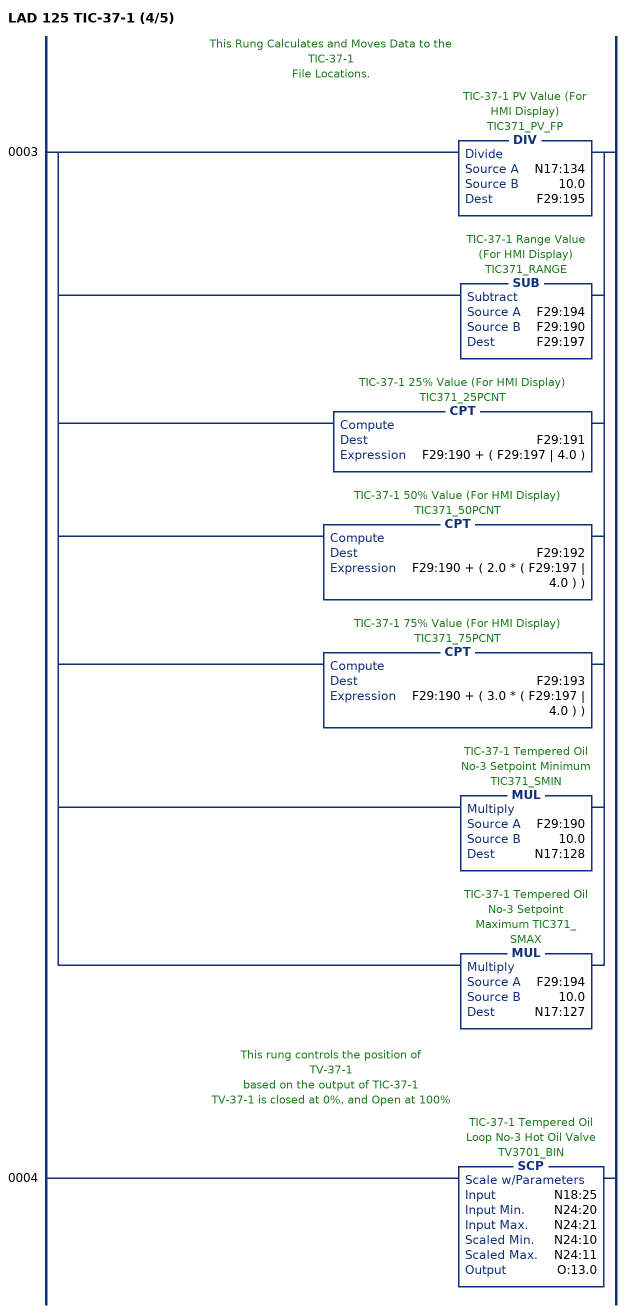
% Rung: 3 %
% This Rung Calculates and Moves Data to the
% TIC-37-1
% File Locations. %
SOR BST DIV N17:134 10.0 F29:195 NXB SUB F29:194 F29:190 F29:197 NXB CPT F29:191 " F29:190 + ( F29:197 | 4.0 ) " NXB CPT F29:192 " F29:190 + ( 2.0 * ( F29:197 | 4.0 ) ) " NXB CPT F29:193 " F29:190 + ( 3.0 * ( F29:197 | 4.0 ) ) " NXB MUL F29:190 10.0 N17:128 NXB MUL F29:194 10.0 N17:127 BND EOR
%   N17:134  TIC371_PV  "TIC-37-1 Tempered Oil No-3 Scaled Process Variable" %
%   F29:195  TIC371_PV_FP  "TIC-37-1 PV Value (For HMI Display)" %
%   F29:194  TIC371_MAX  "TIC-37-1 100% Value (For HMI Display)" %
%   F29:190  TIC371_MIN  "TIC-37-1 0% Value (For HMI Display)" %
%   F29:197  TIC371_RANGE  "TIC-37-1 Range Value (For HMI Display)" %
%   F29:191  TIC371_25PCNT  "TIC-37-1 25% Value (For HMI Display)" %
%   F29:192  TIC371_50PCNT  "TIC-37-1 50% Value (For HMI Display)" %
%   F29:193  TIC371_75PCNT  "TIC-37-1 75% Value (For HMI Display)" %
%   N17:128  TIC371_SMIN  "TIC-37-1 Tempered Oil No-3 Setpoint Minimum" %
%   N17:127  TIC371_SMAX  "TIC-37-1 Tempered Oil No-3 Setpoint Maximum" %
% Rung: 4 %
% This rung controls the position of
% TV-37-1
% based on the output of TIC-37-1
% TV-37-1 is closed at 0%, and Open at 100% %
SOR SCP N18:25 N24:20 N24:21 N24:10 N24:11 O:13.0 EOR
%   N18:25  TIC371_OUT1  "TIC-37-1 Tempered Oil No-3 PID Output Value" %
%   N24:20  PID_MIN  "PID Statement Minimum Value" %
%   N24:21  PID_MAX  "PID Statement Maximum Value" %
%   N24:10  AO_MIN_NO4I  "Analog Output Minimum Value Generates 4 mA DC (To NO4I AO Module)" %
%   N24:11  AO_MAX_NO4I  "Analog Output Maximum Value Generates 20 mA DC (To NO4I AO Module)" %
%   O:13.0  TV3701_BIN  "TIC-37-1 Tempered Oil Loop No-3 Hot Oil Valve" %

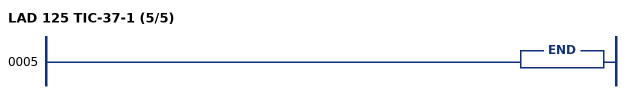
% Rung: 5 %
SOR END EOR

LADDER 126 "TIC-40-1"    % Tempered Oil Loop No-2 Temperature PID Controls %
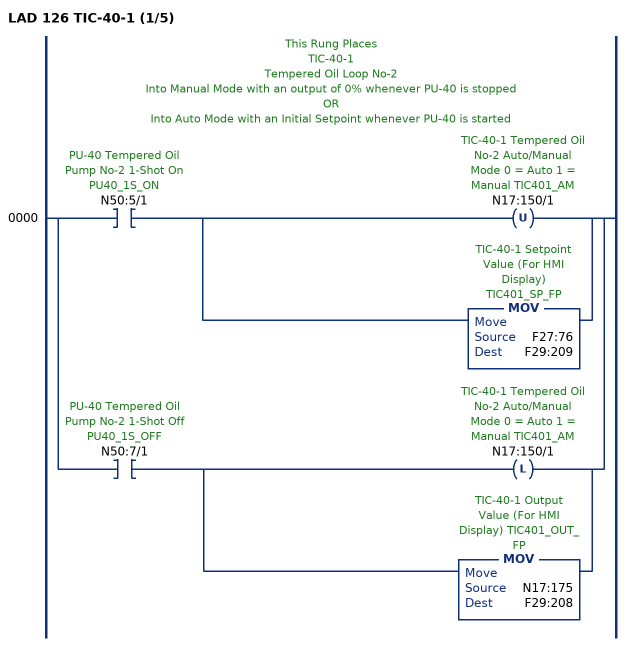
% Rung: 0 %
% This Rung Places
% TIC-40-1
% Tempered Oil Loop No-2
% Into Manual Mode with an output of 0% whenever PU-40 is stopped
% OR
% Into Auto Mode with an Initial Setpoint whenever PU-40 is started %
SOR BST XIC N50:5/1 BST OTU N17:150/1 NXB MOV F27:76 F29:209 BND NXB XIC N50:7/1 BST OTL N17:150/1 NXB MOV N17:175 F29:208 BND BND EOR
%   N50:5/1  PU40_1S_ON  "PU-40 Tempered Oil Pump No-2 1-Shot On" %
%   N17:150/1  TIC401_AM  "TIC-40-1 Tempered Oil No-2 Auto/Manual Mode 0 = Auto 1 = Manual" %
%   F27:76  TIC401_INIT_SP  "TIC-40-1 Initial Temperature Setpoint" %
%   F29:209  TIC401_SP_FP  "TIC-40-1 Setpoint Value (For HMI Display)" %
%   N50:7/1  PU40_1S_OFF  "PU-40 Tempered Oil Pump No-2 1-Shot Off" %
%   N17:175  TIC401_OFF_OUTPUT  "TIC-40-1 Output When PU-13 Is Off" %
%   F29:208  TIC401_OUT_FP  "TIC-40-1 Output Value (For HMI Display)" %

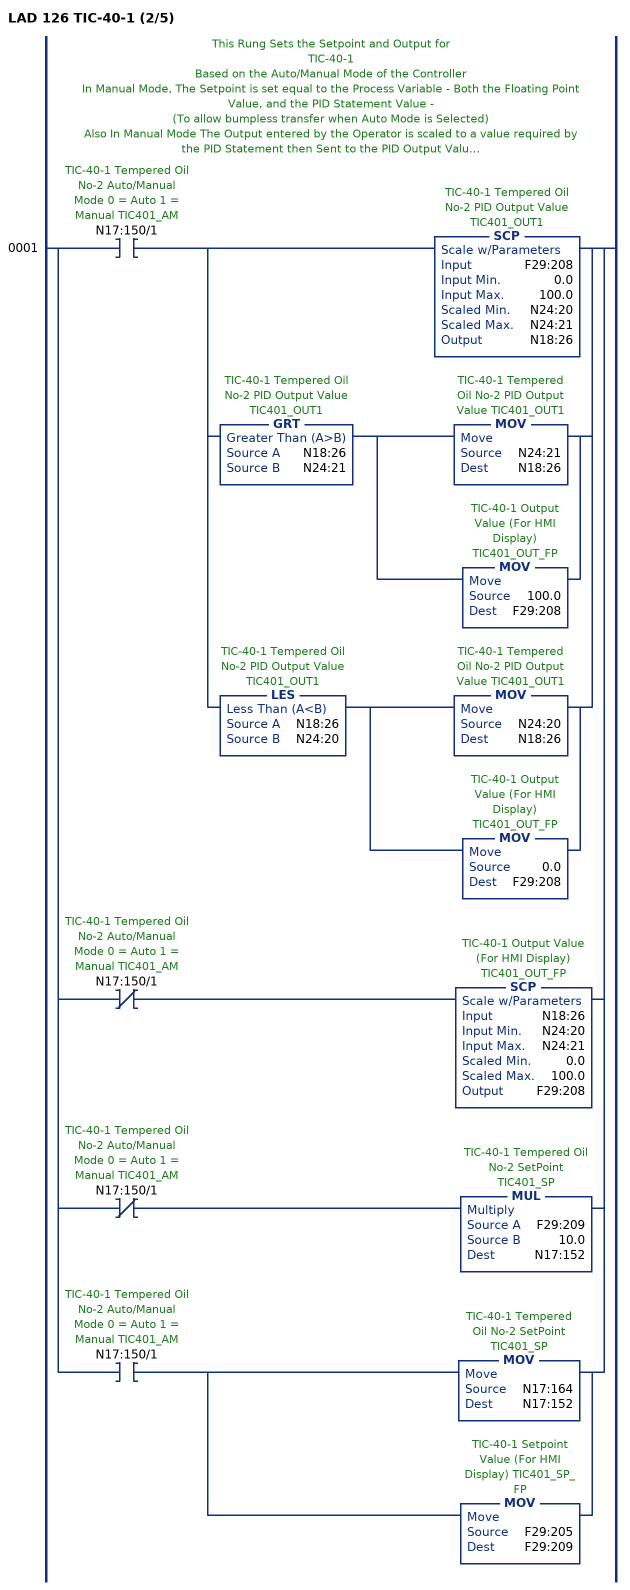
% Rung: 1 %
% This Rung Sets the Setpoint and Output for
% TIC-40-1
% Based on the Auto/Manual Mode of the Controller
% In Manual Mode, The Setpoint is set equal to the Process Variable - Both the Floating Point Value, and the PID Statement Value -
% (To allow bumpless transfer when Auto Mode is Selected)
% Also In Manual Mode The Output entered by the Operator is scaled to a value required by the PID Statement then Sent to the PID Output Value
% 
% In Auto Mode, The Setpoint is Entered by the Operator from Any HMI terminal, Multiplied by 10, and placed in the PID Statement's Setpoint Location
% Also In Auto Mode, the Output (used by the Operator) is set equal to the actual value of the pID statement
% (To allow bumpless transfer when Manual Mode is Selected) %
SOR BST XIC N17:150/1 BST SCP F29:208 0.0 100.0 N24:20 N24:21 N18:26 NXB GRT N18:26 N24:21 BST MOV N24:21 N18:26 NXB MOV 100.0 F29:208 BND NXB LES N18:26 N24:20 BST MOV N24:20 N18:26 NXB MOV 0.0 F29:208 BND BND NXB XIO N17:150/1 SCP N18:26 N24:20 N24:21 0.0 100.0 F29:208 NXB XIO N17:150/1 MUL F29:209 10.0 N17:152 NXB XIC N17:150/1 BST MOV N17:164 N17:152 NXB MOV F29:205 F29:209 BND BND EOR
%   N17:150/1  TIC401_AM  "TIC-40-1 Tempered Oil No-2 Auto/Manual Mode 0 = Auto 1 = Manual" %
%   F29:208  TIC401_OUT_FP  "TIC-40-1 Output Value (For HMI Display)" %
%   N24:20  PID_MIN  "PID Statement Minimum Value" %
%   N24:21  PID_MAX  "PID Statement Maximum Value" %
%   N18:26  TIC401_OUT1  "TIC-40-1 Tempered Oil No-2 PID Output Value" %
%   F29:209  TIC401_SP_FP  "TIC-40-1 Setpoint Value (For HMI Display)" %
%   N17:152  TIC401_SP  "TIC-40-1 Tempered Oil No-2 SetPoint" %
%   N17:164  TIC401_PV  "TIC-40-1 Tempered Oil No-2 Scaled Process Variable" %
%   F29:205  TIC401_PV_FP  "TIC-40-1 PV Value (For HMI Display)" %

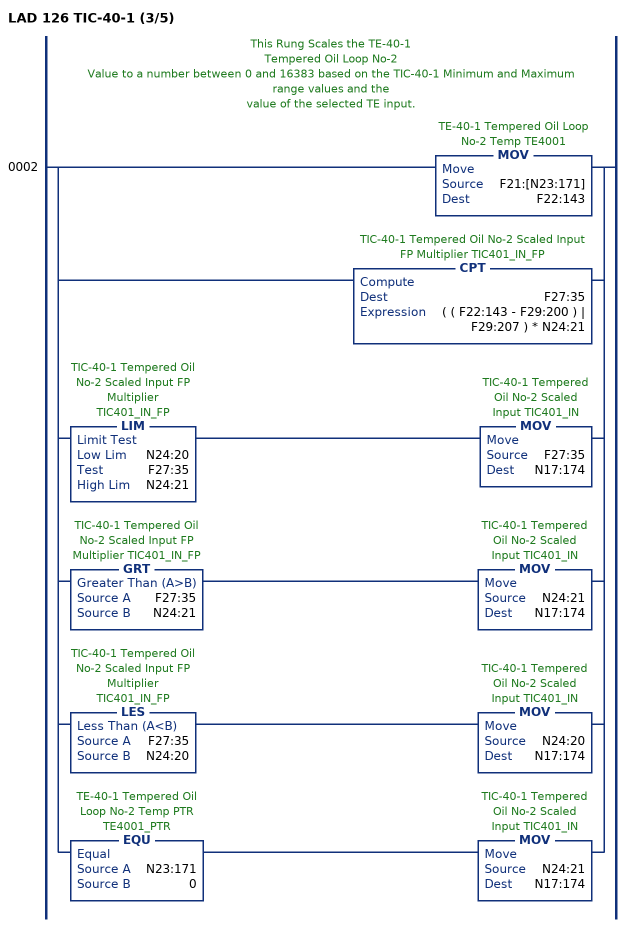
% Rung: 2 %
% This Rung Scales the TE-40-1
% Tempered Oil Loop No-2
% Value to a number between 0 and 16383 based on the TIC-40-1 Minimum and Maximum range values and the
% value of the selected TE input. %
SOR BST MOV F21:[N23:171] F22:143 NXB CPT F27:35 " ( ( F22:143 - F29:200 ) | F29:207 ) * N24:21 " NXB LIM N24:20 F27:35 N24:21 MOV F27:35 N17:174 NXB GRT F27:35 N24:21 MOV N24:21 N17:174 NXB LES F27:35 N24:20 MOV N24:20 N17:174 NXB EQU N23:171 0 MOV N24:21 N17:174 BND EOR
%   N23:171  TE4001_PTR  "TE-40-1 Tempered Oil Loop No-2 Temp PTR" %
%   F22:143  TE4001  "TE-40-1 Tempered Oil Loop No-2 Temp" %
%   F27:35  TIC401_IN_FP  "TIC-40-1 Tempered Oil No-2 Scaled Input FP Multiplier" %
%   F29:200  TIC401_MIN  "TIC-40-1 0% Value (For HMI Display)" %
%   F29:207  TIC401_RANGE  "TIC-40-1 Range Value (For HMI Display)" %
%   N24:21  PID_MAX  "PID Statement Maximum Value" %
%   N24:20  PID_MIN  "PID Statement Minimum Value" %
%   N17:174  TIC401_IN  "TIC-40-1 Tempered Oil No-2 Scaled Input" %

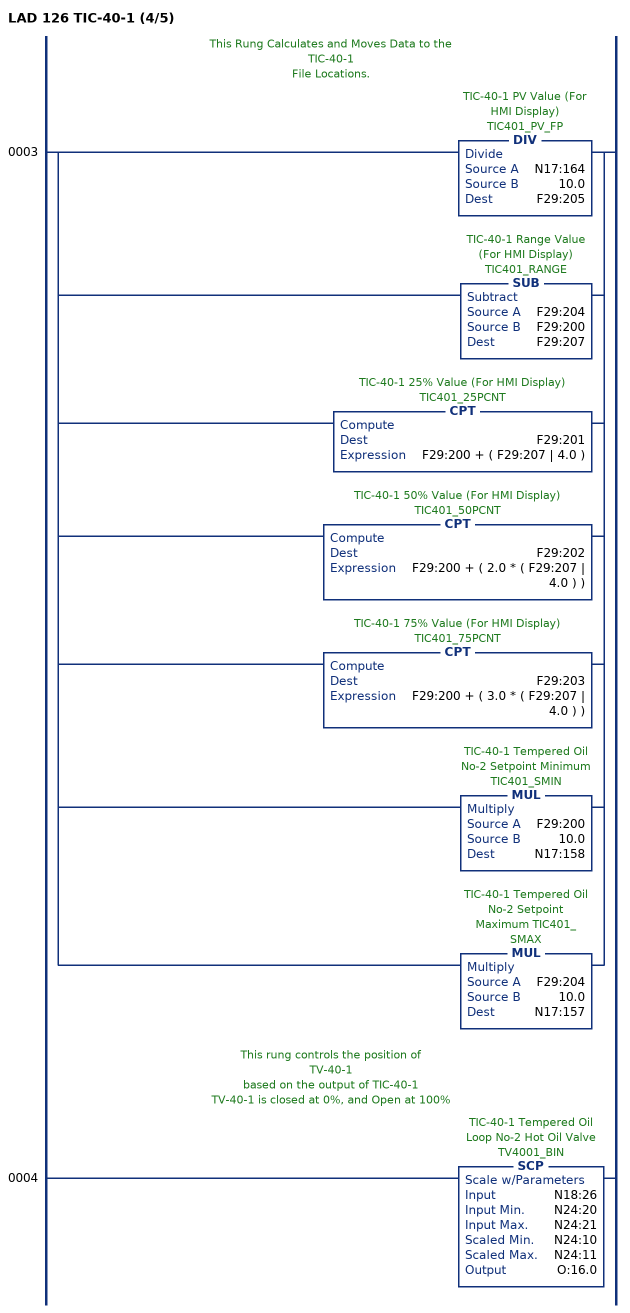
% Rung: 3 %
% This Rung Calculates and Moves Data to the
% TIC-40-1
% File Locations. %
SOR BST DIV N17:164 10.0 F29:205 NXB SUB F29:204 F29:200 F29:207 NXB CPT F29:201 " F29:200 + ( F29:207 | 4.0 ) " NXB CPT F29:202 " F29:200 + ( 2.0 * ( F29:207 | 4.0 ) ) " NXB CPT F29:203 " F29:200 + ( 3.0 * ( F29:207 | 4.0 ) ) " NXB MUL F29:200 10.0 N17:158 NXB MUL F29:204 10.0 N17:157 BND EOR
%   N17:164  TIC401_PV  "TIC-40-1 Tempered Oil No-2 Scaled Process Variable" %
%   F29:205  TIC401_PV_FP  "TIC-40-1 PV Value (For HMI Display)" %
%   F29:204  TIC401_MAX  "TIC-40-1 100% Value (For HMI Display)" %
%   F29:200  TIC401_MIN  "TIC-40-1 0% Value (For HMI Display)" %
%   F29:207  TIC401_RANGE  "TIC-40-1 Range Value (For HMI Display)" %
%   F29:201  TIC401_25PCNT  "TIC-40-1 25% Value (For HMI Display)" %
%   F29:202  TIC401_50PCNT  "TIC-40-1 50% Value (For HMI Display)" %
%   F29:203  TIC401_75PCNT  "TIC-40-1 75% Value (For HMI Display)" %
%   N17:158  TIC401_SMIN  "TIC-40-1 Tempered Oil No-2 Setpoint Minimum" %
%   N17:157  TIC401_SMAX  "TIC-40-1 Tempered Oil No-2 Setpoint Maximum" %
% Rung: 4 %
% This rung controls the position of
% TV-40-1
% based on the output of TIC-40-1
% TV-40-1 is closed at 0%, and Open at 100% %
SOR SCP N18:26 N24:20 N24:21 N24:10 N24:11 O:16.0 EOR
%   N18:26  TIC401_OUT1  "TIC-40-1 Tempered Oil No-2 PID Output Value" %
%   N24:20  PID_MIN  "PID Statement Minimum Value" %
%   N24:21  PID_MAX  "PID Statement Maximum Value" %
%   N24:10  AO_MIN_NO4I  "Analog Output Minimum Value Generates 4 mA DC (To NO4I AO Module)" %
%   N24:11  AO_MAX_NO4I  "Analog Output Maximum Value Generates 20 mA DC (To NO4I AO Module)" %
%   O:16.0  TV4001_BIN  "TIC-40-1 Tempered Oil Loop No-2 Hot Oil Valve" %

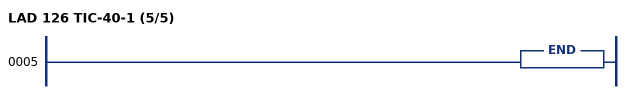
% Rung: 5 %
SOR END EOR

LADDER 131 "LIC-22-1"    % Level Control No-1 PID Controls %
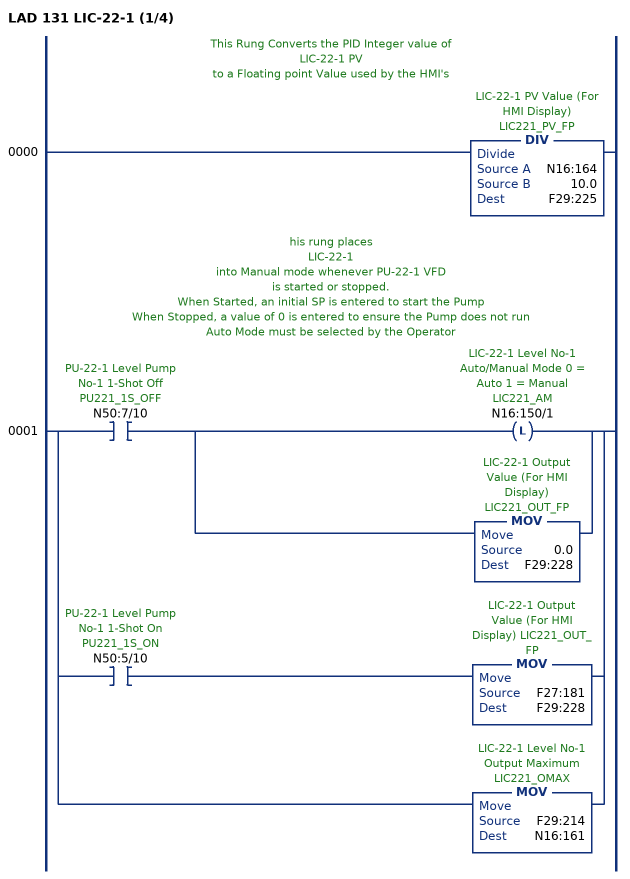
% Rung: 0 %
% This Rung Converts the PID Integer value of
% LIC-22-1 PV
% to a Floating point Value used by the HMI's %
SOR DIV N16:164 10.0 F29:225 EOR
%   N16:164  LIC221_PV  "LIC-22-1 Level No-1 Scaled Process Variable" %
%   F29:225  LIC221_PV_FP  "LIC-22-1 PV Value (For HMI Display)" %
% Rung: 1 %
% his rung places
% LIC-22-1
% into Manual mode whenever PU-22-1 VFD
% is started or stopped.
% When Started, an initial SP is entered to start the Pump
% When Stopped, a value of 0 is entered to ensure the Pump does not run
% Auto Mode must be selected by the Operator %
SOR BST XIC N50:7/10 BST OTL N16:150/1 NXB MOV 0.0 F29:228 BND NXB XIC N50:5/10 MOV F27:181 F29:228 NXB MOV F29:214 N16:161 BND EOR
%   N50:7/10  PU221_1S_OFF  "PU-22-1 Level Pump No-1 1-Shot Off" %
%   N16:150/1  LIC221_AM  "LIC-22-1 Level No-1 Auto/Manual Mode 0 = Auto 1 = Manual" %
%   F29:228  LIC221_OUT_FP  "LIC-22-1 Output Value (For HMI Display)" %
%   N50:5/10  PU221_1S_ON  "PU-22-1 Level Pump No-1 1-Shot On" %
%   F27:181  SIC221_INIT_SP  "SIC-22-1 Initial Speed Setpoint (Hz)" %
%   F29:214  SIC221_MAX  "SIC-22-1 PU-22-1 Level Pump No-1 Freq at 100% Value (For HMI Display)" %
%   N16:161  LIC221_OMAX  "LIC-22-1 Level No-1 Output Maximum" %

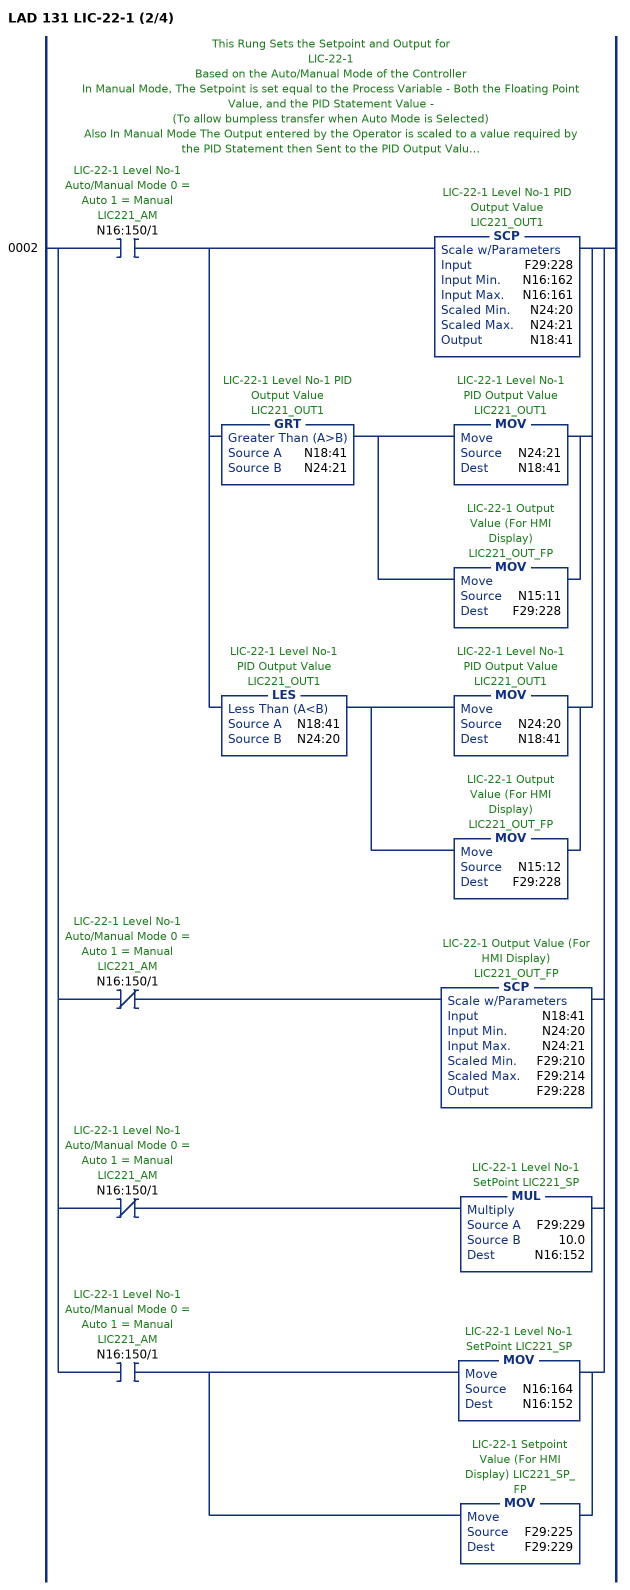
% Rung: 2 %
% This Rung Sets the Setpoint and Output for
% LIC-22-1
% Based on the Auto/Manual Mode of the Controller
% In Manual Mode, The Setpoint is set equal to the Process Variable - Both the Floating Point Value, and the PID Statement Value -
% (To allow bumpless transfer when Auto Mode is Selected)
% Also In Manual Mode The Output entered by the Operator is scaled to a value required by the PID Statement then Sent to the PID Output Value
% 
% In Auto Mode, The Setpoint is Entered by the Operator from Any HMI terminal, Multiplied by 10, and placed in the PID Statement's Setpoint Location
% Also In Auto Mode, the Output (used by the Operator) is set equal to the actual value of the pID statement
% (To allow bumpless transfer when Manual Mode is Selected) %
SOR BST XIC N16:150/1 BST SCP F29:228 N16:162 N16:161 N24:20 N24:21 N18:41 NXB GRT N18:41 N24:21 BST MOV N24:21 N18:41 NXB MOV N15:11 F29:228 BND NXB LES N18:41 N24:20 BST MOV N24:20 N18:41 NXB MOV N15:12 F29:228 BND BND NXB XIO N16:150/1 SCP N18:41 N24:20 N24:21 F29:210 F29:214 F29:228 NXB XIO N16:150/1 MUL F29:229 10.0 N16:152 NXB XIC N16:150/1 BST MOV N16:164 N16:152 NXB MOV F29:225 F29:229 BND BND EOR
%   N16:150/1  LIC221_AM  "LIC-22-1 Level No-1 Auto/Manual Mode 0 = Auto 1 = Manual" %
%   F29:228  LIC221_OUT_FP  "LIC-22-1 Output Value (For HMI Display)" %
%   N16:162  LIC221_OMIN  "LIC-22-1 Level No-1 Output Minimum" %
%   N16:161  LIC221_OMAX  "LIC-22-1 Level No-1 Output Maximum" %
%   N24:20  PID_MIN  "PID Statement Minimum Value" %
%   N24:21  PID_MAX  "PID Statement Maximum Value" %
%   N18:41  LIC221_OUT1  "LIC-22-1 Level No-1 PID Output Value" %
%   N15:11  FIC211_OMAX  "FIC-21-1 Feed Flow No-1 Output Maximum" %
%   N15:12  FIC211_OMIN  "FIC-21-1 Feed Flow No-1 Output Minimum" %
%   F29:210  SIC221_MIN  "SIC-22-1 PU-22-1 Level Pump No-1 Speed 0% Value (For HMI Display)" %
%   F29:214  SIC221_MAX  "SIC-22-1 PU-22-1 Level Pump No-1 Freq at 100% Value (For HMI Display)" %
%   F29:229  LIC221_SP_FP  "LIC-22-1 Setpoint Value (For HMI Display)" %
%   N16:152  LIC221_SP  "LIC-22-1 Level No-1 SetPoint" %
%   N16:164  LIC221_PV  "LIC-22-1 Level No-1 Scaled Process Variable" %
%   F29:225  LIC221_PV_FP  "LIC-22-1 PV Value (For HMI Display)" %

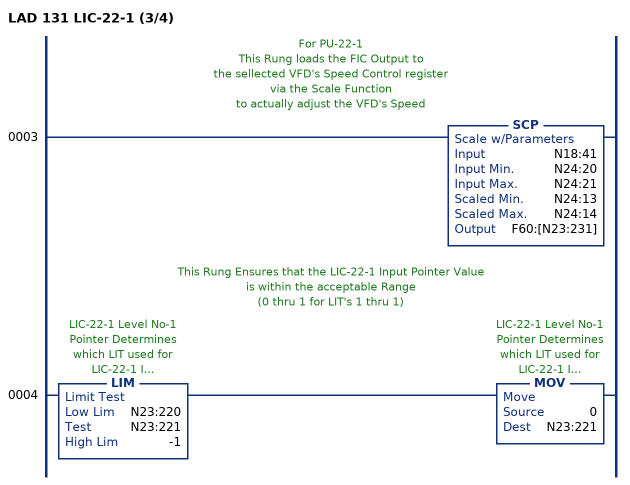
% Rung: 3 %
% For PU-22-1
% This Rung loads the FIC Output to
% the sellected VFD's Speed Control register
% via the Scale Function
% to actually adjust the VFD's Speed %
SOR SCP N18:41 N24:20 N24:21 N24:13 N24:14 F60:[N23:231] EOR
%   N18:41  LIC221_OUT1  "LIC-22-1 Level No-1 PID Output Value" %
%   N24:20  PID_MIN  "PID Statement Minimum Value" %
%   N24:21  PID_MAX  "PID Statement Maximum Value" %
%   N24:13  AO_MIN_OE4  "Analog Output Minimum Value Generates 4 mA DC (To OE4 AO Module)" %
%   N24:14  AO_MAX_OE4  "Analog Output Maximum Value Generates 20 mA DC (To OE4 AO Module)" %
%   N23:231  LIC221_OUT_PTR  "LIC-22-1 Level No-1 Output Pointer Determines which VFD is controled by LIC" %
% Rung: 4 %
% This Rung Ensures that the LIC-22-1 Input Pointer Value
% is within the acceptable Range
% (0 thru 1 for LIT's 1 thru 1) %
SOR LIM N23:220 N23:221 -1 MOV 0 N23:221 EOR
%   N23:220  MAX_LIT_ALLOWED_1  "Maximum Number of LITs Available Plus 1" %
%   N23:221  LIC221_IN_PTR  "LIC-22-1 Level No-1 Pointer Determines which LIT used for LIC-22-1 In" %

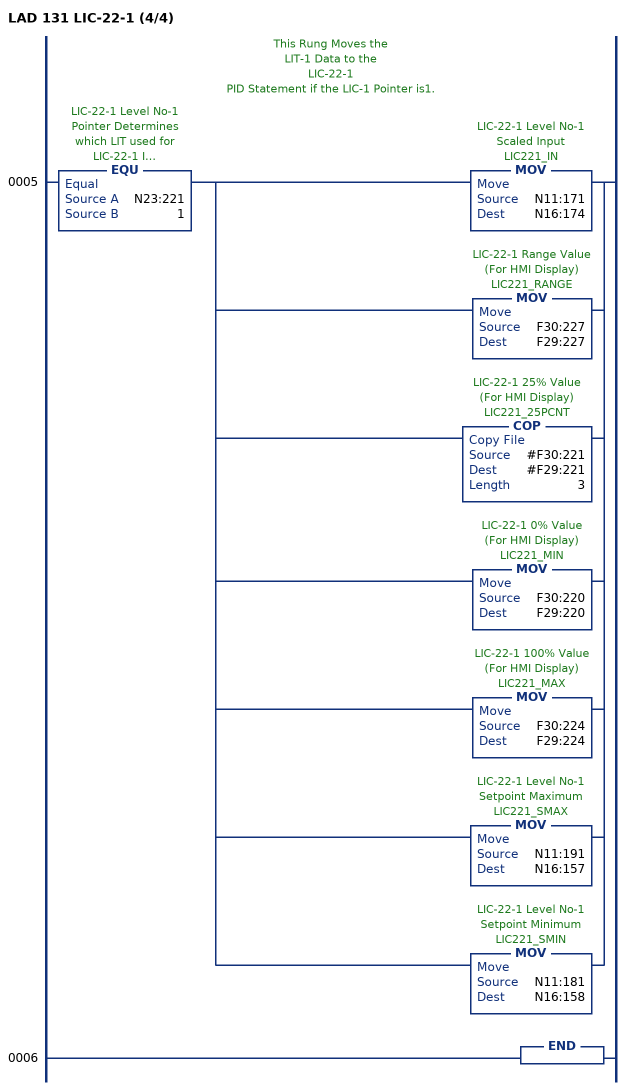
% Rung: 5 %
% This Rung Moves the
% LIT-1 Data to the
% LIC-22-1
% PID Statement if the LIC-1 Pointer is1. %
SOR EQU N23:221 1 BST MOV N11:171 N16:174 NXB MOV F30:227 F29:227 NXB COP #F30:221 #F29:221 3 NXB MOV F30:220 F29:220 NXB MOV F30:224 F29:224 NXB MOV N11:191 N16:157 NXB MOV N11:181 N16:158 BND EOR
%   N23:221  LIC221_IN_PTR  "LIC-22-1 Level No-1 Pointer Determines which LIT used for LIC-22-1 In" %
%   N11:171  LIT01_PID_IN  "LIT-1 Level Transmitter No-1 PID Statement Input Value" %
%   N16:174  LIC221_IN  "LIC-22-1 Level No-1 Scaled Input" %
%   F30:227  LIT01_RANGE  "LIT-1 Range (%) MAX - MIN" %
%   F29:227  LIC221_RANGE  "LIC-22-1 Range Value (For HMI Display)" %
%   F30:221  LIT01_25PCNT_VALUE  "LIT-1 25% Range Value For HMI Display (%)" %
%   F29:221  LIC221_25PCNT  "LIC-22-1 25% Value (For HMI Display)" %
%   F30:220  LIT01_MIN  "LIT-1 Minimum Value (%)" %
%   F29:220  LIC221_MIN  "LIC-22-1 0% Value (For HMI Display)" %
%   F30:224  LIT01_MAX  "LIT-1 Maximum Value (%)" %
%   F29:224  LIC221_MAX  "LIC-22-1 100% Value (For HMI Display)" %
%   N11:191  LIT01_PID_MAX  "LIT-1 Level Transmitter No-1 PID Statement Maximum Input Value" %
%   N16:157  LIC221_SMAX  "LIC-22-1 Level No-1 Setpoint Maximum" %
%   N11:181  LIT01_PID_MIN  "LIT-1 Level Transmitter No-1 PID Statement Minimum Input Value" %
%   N16:158  LIC221_SMIN  "LIC-22-1 Level No-1 Setpoint Minimum" %
% Rung: 6 %
SOR END EOR

LADDER 132 "TOTALIZER"
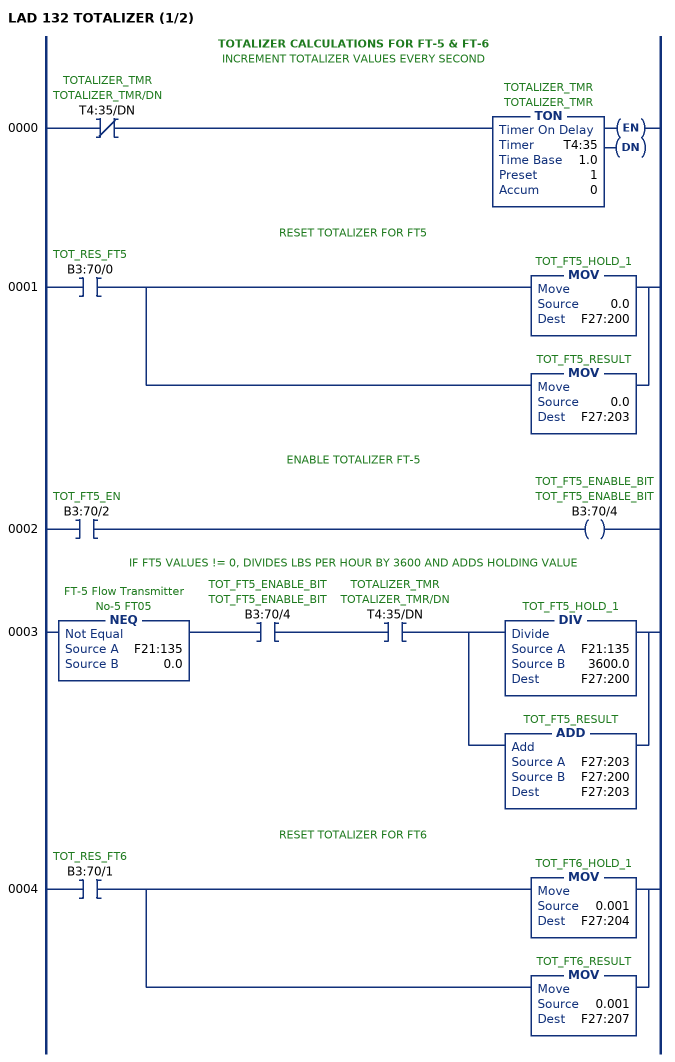
% Rung: 0 %
% TITLE: TOTALIZER CALCULATIONS FOR FT-5 & FT-6 %
% INCREMENT TOTALIZER VALUES EVERY SECOND %
SOR XIO T4:35/DN TON T4:35 1.0 1 0 EOR
%   T4:35  TOTALIZER_TMR  "TOTALIZER_TMR" %
% Rung: 1 %
% RESET TOTALIZER FOR FT5 %
SOR XIC B3:70/0 BST MOV 0.0 F27:200 NXB MOV 0.0 F27:203 BND EOR
%   B3:70/0  TOT_RES_FT5 %
%   F27:200  TOT_FT5_HOLD_1 %
%   F27:203  TOT_FT5_RESULT %
% Rung: 2 %
% ENABLE TOTALIZER FT-5 %
SOR XIC B3:70/2 OTE B3:70/4 EOR
%   B3:70/2  TOT_FT5_EN %
%   B3:70/4  TOT_FT5_ENABLE_BIT  "TOT_FT5_ENABLE_BIT" %
% Rung: 3 %
% IF FT5 VALUES != 0, DIVIDES LBS PER HOUR BY 3600 AND ADDS HOLDING VALUE %
SOR NEQ F21:135 0.0 XIC B3:70/4 XIC T4:35/DN BST DIV F21:135 3600.0 F27:200 NXB ADD F27:203 F27:200 F27:203 BND EOR
%   F21:135  FT05  "FT-5 Flow Transmitter No-5" %
%   B3:70/4  TOT_FT5_ENABLE_BIT  "TOT_FT5_ENABLE_BIT" %
%   T4:35  TOTALIZER_TMR  "TOTALIZER_TMR" %
%   F27:200  TOT_FT5_HOLD_1 %
%   F27:203  TOT_FT5_RESULT %
% Rung: 4 %
% RESET TOTALIZER FOR FT6 %
SOR XIC B3:70/1 BST MOV 0.001 F27:204 NXB MOV 0.001 F27:207 BND EOR
%   B3:70/1  TOT_RES_FT6 %
%   F27:204  TOT_FT6_HOLD_1 %
%   F27:207  TOT_FT6_RESULT %

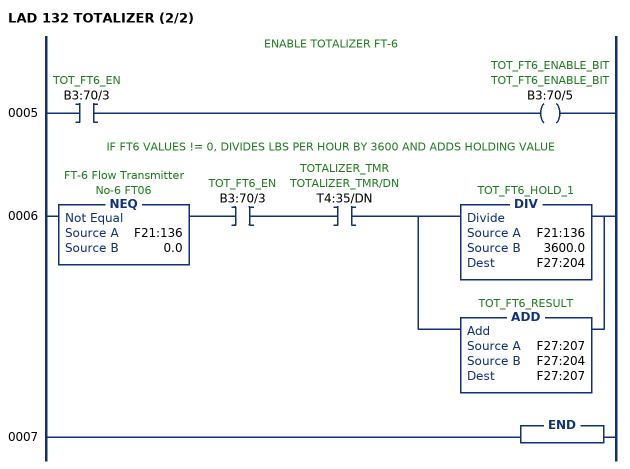
% Rung: 5 %
% ENABLE TOTALIZER FT-6 %
SOR XIC B3:70/3 OTE B3:70/5 EOR
%   B3:70/3  TOT_FT6_EN %
%   B3:70/5  TOT_FT6_ENABLE_BIT  "TOT_FT6_ENABLE_BIT" %
% Rung: 6 %
% IF FT6 VALUES != 0, DIVIDES LBS PER HOUR BY 3600 AND ADDS HOLDING VALUE %
SOR NEQ F21:136 0.0 XIC B3:70/3 XIC T4:35/DN BST DIV F21:136 3600.0 F27:204 NXB ADD F27:207 F27:204 F27:207 BND EOR
%   F21:136  FT06  "FT-6 Flow Transmitter No-6" %
%   B3:70/3  TOT_FT6_EN %
%   T4:35  TOTALIZER_TMR  "TOTALIZER_TMR" %
%   F27:204  TOT_FT6_HOLD_1 %
%   F27:207  TOT_FT6_RESULT %
% Rung: 7 %
SOR END EOR

OTHER DOCUMENTED ADDRESSES
  B3:0/0  ALWAYS_OFF  "Bit Used for HMI PB States Always = 0"
  B3:10  ALARM_ITEMS  "Alarm Items (Horns, etc)"
  B3:19/0  AFI
  DFILE:0  "OUTPUT"
  DFILE:1  "INPUT"
  DFILE:2  "STATUS"
  DFILE:3  "BINARY"
  DFILE:4  "TIMER"
  DFILE:5  "COUNTER"
  DFILE:6  "CONTROL"
  DFILE:7  "INTEGER"
  DFILE:8  "FLOAT"
  DFILE:9  "FLOW_AVGS Flow Rates Used in C alculating 5 Minute Averages"
  DFILE:11  "AI INTEGER Integer Data for All Inputs (TE's, PT's and FT's)"
  DFILE:12  "RIO DATA Remote I/O Data"
  DFILE:13  "TE SETUP TE Setup Data"
  DFILE:14  "SETPOINTS Setpoints for variou s Alarms, trips, etc"
  DFILE:15  "PID 1 OF 3 PID Statement Contro ls File No-1"
  DFILE:16  "PID 2 OF 3 PID Statement Contro ls File No-2"
  DFILE:17  "PID 3 OF 3 PID Statement Contro ls File No-3"
  DFILE:18  "PID OUTPUT Outputs from All PID Statements"
  DFILE:20  "PANELVIEW Info From/to PanelVi ew HMIs"
  DFILE:21  "AI REAL"
  DFILE:22  "AI BY TAG"
  DFILE:23  "AI PTRS"
  DFILE:24  "FIXED INTS Fixed Integer Values"
  DFILE:25  "VAR INTS Variable Integer Val ues"
  DFILE:26  "FIXEDREAL1 Fixed Real (Floating Point) Data 1 of 2"
  DFILE:27  "VAR REAL Variable Real (Float inf Point) Data"
  DFILE:28  "FLOW AVGS Flow Data used to Ca lculate 5 Minute Ave erages"
  DFILE:29  "PID PCNTS1 PID Statement 0, 25, 50, 75 & 100% Value s"
  DFILE:30  "FIXEDREAL2 Fixed Real (Floating Point) Data 2 of 2"
  DFILE:31  "PID PCNTS2"
  DFILE:50  "CNTL BITS Control Bits for all Motors, Contacters, Etc"
  DFILE:51  "ALARM TMRS Alarm Timers"
  DFILE:52  "ALARM SPS Alarm Setpoints"
  DFILE:60  "VFD TABLE Provide sequencial t able for VFD outputs"
  DFILE:61  "VFD BITS Provide seq table fo r VFD Contrl & Statu s Bits"
  DFILE:62  "VFD AMPS VFD Amps"
  DFILE:63  "VFD HP Motor and VFD Hps"
  DFILE:100  "CH0 Diag"
  DFILE:101  "CH1 Diag"
  DFILE:102  "I:2 DATA"
  DFILE:103  "I:3 DATA"
  DFILE:104  "I:4 DATA"
  DFILE:105  "I:5 DATA"
  DFILE:106  "I:6 DATA"
  DFILE:107  "I:7 DATA"
  DFILE:108  "I:8 DATA"
  DFILE:109  "I:9 DATA"
  DFILE:110  "I:10 DATA"
  DFILE:111  "I:11 DATA"
  DFILE:112  "I:12 DATA"
  DFILE:117  "I:17 DATA"
  DFILE:118  "I:18 DATA"
  DFILE:119  "I:19 DATA"
  DFILE:120  "I:20 DATA"
  DFILE:121  "I:21 DATA"
  DFILE:122  "I:22 DATA"
  DFILE:201  "FT1 AVGS Average FT-1 Values"
  DFILE:202  "FT2 AVGS Average FT-2 Values"
  DFILE:203  "FT3 AVGS Average FT-3 Values"
  DFILE:204  "FT4 AVGS Average FT-4 Values"
  DFILE:205  "FT5 AVGS Average FT-5 Values"
  DFILE:206  "FT6 AVGS Average FT-6 Values"
  DFILE:207  "O:7 DATA"
  DFILE:208  "O:8 DATA"
  DFILE:209  "O:9 DATA"
  DFILE:210  "O:10 DATA"
  DFILE:211  "O:11 DATA"
  DFILE:212  "O:12 DATA"
  DFILE:213  "O:13 DATA"
  DFILE:214  "O:14 DATA"
  DFILE:215  "O:16 DATA"
  DFILE:216  "O:16 DATA"
  DFILE:218  "O:18 DATA"
  DFILE:223  "O:23 DATA"
  DFILE:224  "O:24 DATA"
  DFILE:225  "O:25 DATA"
  F8:0  "Dummy"
  F21:1  TE01_REAL  "Real Value (Floating Point) for TE-1"
  F21:2  TE02_REAL  "Real Value (Floating Point) for TE-2"
  F21:3  TE03_REAL  "Real Value (Floating Point) for TE-3"
  F21:4  TE04_REAL  "Real Value (Floating Point) for TE-4"
  F21:5  TE05_REAL  "Real Value (Floating Point) for TE-5"
  F21:6  TE06_REAL  "Real Value (Floating Point) for TE-6"
  F21:7  TE07_REAL  "Real Value (Floating Point) for TE-7"
  F21:8  TE08_REAL  "Real Value (Floating Point) for TE-8"
  F21:9  TE09_REAL  "Real Value (Floating Point) for TE-9"
  F21:10  TE10_REAL  "Real Value (Floating Point) for TE-10"
  F21:11  TE11_REAL  "Real Value (Floating Point) for TE-11"
  F21:12  TE12_REAL  "Real Value (Floating Point) for TE-12"
  F21:13  TE13_REAL  "Real Value (Floating Point) for TE-13"
  F21:14  TE14_REAL  "Real Value (Floating Point) for TE-14"
  F21:15  TE15_REAL  "Real Value (Floating Point) for TE-15"
  F21:16  TE16_REAL  "Real Value (Floating Point) for TE-16"
  F21:17  TE17_REAL  "Real Value (Floating Point) for TE-17"
  F21:18  TE18_REAL  "Real Value (Floating Point) for TE-18"
  F21:19  TE19_REAL  "Real Value (Floating Point) for TE-19"
  F21:20  TE20_REAL  "Real Value (Floating Point) for TE-20"
  F21:21  TE21_REAL  "Real Value (Floating Point) for TE-21"
  F21:22  TE22_REAL  "Real Value (Floating Point) for TE-22"
  F21:23  TE23_REAL  "Real Value (Floating Point) for TE-23"
  F21:24  TE24_REAL  "Real Value (Floating Point) for TE-24"
  F21:25  TE25_REAL  "Real Value (Floating Point) for TE-25"
  F21:26  TE26_REAL  "Real Value (Floating Point) for TE-26"
  F21:27  TE27_REAL  "Real Value (Floating Point) for TE-27"
  F21:28  TE28_REAL  "Real Value (Floating Point) for TE-28"
  F21:29  TE29_REAL  "Real Value (Floating Point) for TE-29"
  F21:30  TE30_REAL  "Real Value (Floating Point) for TE-30"
  F21:31  TE31_REAL  "Real Value (Floating Point) for TE-31"
  F21:32  TE32_REAL  "Real Value (Floating Point) for TE-32"
  F21:33  TE33_REAL  "Real Value (Floating Point) for TE-33"
  F21:34  TE34_REAL  "Real Value (Floating Point) for TE-34"
  F21:35  TE35_REAL  "Real Value (Floating Point) for TE-35"
  F21:36  TE36_REAL  "Real Value (Floating Point) for TE-36"
  F21:65  FI0101  "FI-1-1 EV-1 Condensor Water Flow via Operator Entry"
  F21:66  FI0201  "FI-2-1 EV-2 Condensor Water Flow via Operator Entry"
  F21:130  FT00  "FT-0 Zero Value for FT Moves"
  F21:202  LIT02  "LIT-2 Level (%) Level Pot No-2"
  F21:203  LIT03  "LIT-3 Level (%) Level Pot No-3"
  F22:14  PT0401  "PT-4-1"
  F22:15  PT0501  "PT-5-1"
  F22:16  PT0601  "PT-6-1"
  F27:201  TOT_FT5_HOLD_2
  F27:205  TOT_FT6_HOLD_2
  F29:2  FIC211_50PCNT  "FIC-21-1 50% Value (For HMI Display)"
  F29:3  FIC211_75PCNT  "FIC-21-1 75% Value (For HMI Display)"
  F29:12  FIC212_50PCNT  "FIC-21-2 50% Value (For HMI Display)"
  F29:13  FIC212_75PCNT  "FIC-21-2 75% Value (For HMI Display)"
  F29:22  FIC213_50PCNT  "FIC-21-3 50% Value (For HMI Display)"
  F29:23  FIC213_75PCNT  "FIC-21-3 75% Value (For HMI Display)"
  F29:32  FIC214_50PCNT  "FIC-21-4 50% Value (For HMI Display)"
  F29:33  FIC214_75PCNT  "FIC-21-4 75% Value (For HMI Display)"
  F29:52  PIC091_50PCNT  "PIC-9-1 50% Value (For HMI Display)"
  F29:53  PIC091_75PCNT  "PIC-9-1 75% Value (For HMI Display)"
  F29:62  PIC101_50PCNT  "PIC-10-1 50% Value (For HMI Display)"
  F29:63  PIC101_75PCNT  "PIC-10-1 75% Value (For HMI Display)"
  F29:72  PIC281_50PCNT  "PIC-28-1 50% Value (For HMI Display)"
  F29:73  PIC281_75PCNT  "PIC-28-1 75% Value (For HMI Display)"
  F29:82  PIC301_50PCNT  "PIC-30-1 50% Value (For HMI Display)"
  F29:83  PIC301_75PCNT  "PIC-30-1 75% Value (For HMI Display)"
  F29:95  SIC301_PV_FP  "SIC-30-1 PU-30 Water Booster Pump Speed PV Value (For HMI Display)"
  F29:98  SIC301_OUT_FP  "SIC-30-1 PU-30 Water Booster Pump Speed Outpu Value (For HMI Display)"
  F29:105  SIC021_PV_FP  "SIC-2-1 EV-2 Rotor Speed PV Value (For HMI Display)"
  F29:106  SIC021_MAX_HZ  "SIC-2-1 EV-2 Rotor Hz at 100% Speed Value (For HMI Display)"
  F29:108  SIC021_OUT_FP  "SIC-2-1 EV-2 Rotor Speed Output Value (For HMI Display)"
  F29:115  SIC031_PV_FP  "SIC-3-1 EV-3 Rotor Speed PV Value (For HMI Display)"
  F29:116  SIC031_MAX_HZ  "SIC-3-1 EV-3 Rotor Hz at 100% Speed Value (For HMI Display)"
  F29:118  SIC031_OUT_FP  "SIC-3-1 EV-3 Rotor Speed Output Value (For HMI Display)"
  F29:125  SIC041_PV_FP  "SIC-4-1 AG-4 Agitator Speed PV Value (For HMI Display)"
  F29:126  SIC041_MAX_HZ  "SIC-4-1 AG-4 Agitator Hz at 100% Speed Value (For HMI Display)"
  F29:128  SIC041_OUT_FP  "SIC-4-1 AG-4 Agitator Speed Output Value (For HMI Display)"
  F29:135  SIC211_PV_FP  "SIC-21-1 PU-21-1 Feed Pump No-1 Speed PV Value (For HMI Display)"
  F29:136  SIC211_MAX_HZ  "SIC-21-1 PU-21-1 Hz at 100% Speed Value (For HMI Display)"
  F29:138  SIC211_OUT_FP  "SIC-21-1 PU-21-1 Feed Pump No-1 Speed Output Value (For HMI Display)"
  F29:145  SIC212_PV_FP  "SIC-21-2 PU-21-2 Feed Pump No-2 Speed PV Value (For HMI Display)"
  F29:146  SIC212_MAX_HZ  "SIC-21-2 PU-21-2 Hz at 100% Speed Value (For HMI Display)"
  F29:148  SIC212_OUT_FP  "SIC-21-2 PU-21-2 Feed Pump No-2 Speed Output Value (For HMI Display)"
  F29:215  SIC221_PV_FP  "SIC-22-1 PU-22-1 Level Pump No-1 Speed PV Value (For HMI Display)"
  F29:216  SIC221_MAX_HZ  "SIC-22-1 PU-22-1 Hz at 100% Speed Value (For HMI Display)"
  F29:218  SIC221_OUT_FP  "SIC-22-1 PU-22-1 Level Pump No-1 Speed Output Value (For HMI Display)"
  F29:222  LIC221_50PCNT  "LIC-22-1 50% Value (For HMI Display)"
  F29:223  LIC221_75PCNT  "LIC-22-1 75% Value (For HMI Display)"
  F30:0  IT021_MIN  "IT-2-1 Minimum Value (Amps)"
  F30:1  IT021_25PCNT_VALUE  "IT-2-1 25% Range Value For HMI Display"
  F30:2  "IT-2-1 50% Range Value For HMI Display"
  F30:55  SIC213_PV_FP  "SIC-21-3 PU-21-3 Feed Pump No-3 Speed PV Value (For HMI Display)"
  F30:56  SIC213_MAX_HZ  "SIC-21-3 PU-21-3 Hz at 100% Speed Value (For HMI Display)"
  F30:58  SIC213_OUT_FP  "SIC-21-3 PU-21-3 Feed Pump No-3 Speed Output Value (For HMI Display)"
  F30:65  SIC214_PV_FP  "SIC-21-4 PU-21-4 Feed Pump No-4 Speed PV Value (For HMI Display)"
  F30:66  SIC214_MAX_HZ  "SIC-21-4 PU-21-4 Hz at 100% Speed Value (For HMI Display)"
  F30:68  SIC214_OUT_FP  "SIC-21-4 PU-21-4 Feed Pump No-4 Speed Output Value (For HMI Display)"
  F30:75  SIC461_PV_FP  "SIC-46-1 PU-46 Flash Evap Circ Pump Speed PV Value (For HMI Display)"
  F30:76  SIC461_MAX_HZ  "SIC-46-1 PU-46-1 Hz at 100% Speed Value (For HMI Display)"
  F30:78  SIC461_OUT_FP  "SIC-46-1 PU-46 Flash Evap Circ Pump Speed Output Value (For HMI Display)"
  F30:85  SIC201_PV_FP  "SIC-20-1 EV-20 Rotor Speed PV Value (For HMI Display)"
  F30:86  SIC201_MAX_HZ  "SIC-20-1 EV-20 Rotor Hz at 100% Speed Value (For HMI Display)"
  F30:88  SIC201_OUT_FP  "SIC-20-1 EV-20 Rotor Speed Output Value (For HMI Display)"
  F30:95  SIC421_PV_FP  "SIC-42-1 EV-42 Rotor Speed PV Value (For HMI Display)"
  F30:96  SIC421_MAX_HZ  "SIC-42-1 EV-42 Rotor Hz at 100% Speed Value (For HMI Display)"
  F30:98  SIC421_OUT_FP  "SIC-42-1 EV-42 Rotor Speed Output Value (For HMI Display)"
  F30:225  "LIC-22-1 PV Value (For HMI Display)"
  F30:228  "LIC-22-1 Level No-1 Output Value (For HMI Display)"
  F30:229  "LIC-22-1 Level No-1 Setpoint Value (For HMI Display)"
  F62:0  VFD_ZERO_AMPS  "VFD Amps when Not Selected DO NOT CHANGE"
  F63:1  VFD01_HP  "VFD01 Horse Power"
  F63:2  VFD02_HP  "VFD02 Horse Power"
  F63:3  VFD03_HP  "VFD03 Horse Power"
  F63:4  VFD04_HP  "VFD04 Horse Power"
  F63:5  VFD05_HP  "VFD05 Horse Power"
  F63:6  VFD06_HP  "VFD06 Horse Power"
  F63:7  VFD07_HP  "VFD07 Horse Power"
  F63:8  VFD08_HP  "VFD08 Horse Power"
  I:7.1  TE02_BIN  "Binary Input data for TE-2"
  I:7.2  TE03_BIN  "Binary Input data for TE-3"
  I:7.3  TE04_BIN  "Binary Input data for TE-4"
  I:8.0  TE05_BIN  "Binary Input data for TE-5"
  I:8.1  TE06_BIN  "Binary Input data for TE-6"
  I:8.2  TE07_BIN  "Binary Input data for TE-7"
  I:8.3  TE08_BIN  "Binary Input data for TE-8"
  I:9.1  TE10_BIN  "Binary Input data for TE-10"
  I:9.2  TE11_BIN  "Binary Input data for TE-11"
  I:9.3  TE12_BIN  "Binary Input data for TE-12"
  I:10.1  TE14_BIN  "Binary Input data for TE-14"
  I:10.2  TE15_BIN  "Binary Input data for TE-15"
  I:10.3  TE16_BIN  "Binary Input data for TE-16"
  I:11.1  TE18_BIN  "Binary Input data for TE-18"
  I:11.2  TE19_BIN  "Binary Input data for TE-19"
  I:11.3  TE20_BIN  "Binary Input data for TE-20"
  I:12.1  TE22_BIN  "Binary Input data for TE-22"
  I:12.2  TE23_BIN  "Binary Input data for TE-23"
  I:12.3  TE24_BIN  "Binary Input data for TE-24"
  I:17.4  PT2601_BIN  "PT-26-1 Binary Input From Transmitter Analog Input Module"
  I:18.1  TE26_BIN  "Binary Input data for TE-26"
  I:18.2  TE27_BIN  "Binary Input data for TE-27"
  I:18.3  TE28_BIN  "Binary Input data for TE-28"
  I:20.0/15  PU27_RUN  "PU-27 Boil Feed Water Pump Running Controled by Boiler"
  M00000:006.100  TE29_36_M_WORD_0  "TE-29 thru TE-36 M-File Address"
  N11:2  TE_02  "Integer data for TE-2"
  N11:3  TE_03  "Integer data for TE-3"
  N11:4  TE_04  "Integer data for TE-4"
  N11:5  TE_05  "Integer data for TE-5"
  N11:6  TE_06  "Integer data for TE-6"
  N11:7  TE_07  "Integer data for TE-7"
  N11:8  TE_08  "Integer data for TE-8"
  N11:10  TE_10  "Integer data for TE-10"
  N11:11  TE_11  "Integer data for TE-11"
  N11:12  TE_12  "Integer data for TE-12"
  N11:14  TE_14  "Integer data for TE-14"
  N11:15  TE_15  "Integer data for TE-15"
  N11:16  TE_16  "Integer data for TE-16"
  N11:18  TE_18  "Integer data for TE-18"
  N11:19  TE_19  "Integer data for TE-19"
  N11:20  TE_20  "Integer data for TE-20"
  N11:22  TE_22  "Integer data for TE-22"
  N11:23  TE_23  "Integer data for TE-23"
  N11:24  TE_24  "Integer data for TE-24"
  N11:26  TE_26  "Integer data for TE-26"
  N11:27  TE_27  "Integer data for TE-27"
  N11:28  TE_28  "Integer data for TE-28"
  N11:30  TE_30  "Integer data for TE-30"
  N11:31  TE_31  "Integer data for TE-31"
  N11:32  TE_32  "Integer data for TE-32"
  N11:33  TE_33  "Integer data for TE-33"
  N11:34  TE_34  "Integer data for TE-34"
  N11:35  TE_35  "Integer data for TE-35"
  N11:36  TE_36  "Integer data for TE-36"
  N12:2  TE30_BIN  "Binary data for TE-30"
  N12:3  TE31_BIN  "Binary data for TE-31"
  N12:4  TE32_BIN  "Binary data for TE-32"
  N12:5  TE33_BIN  "Binary data for TE-33"
  N12:6  TE34_BIN  "Binary data for TE-34"
  N12:7  TE35_BIN  "Binary data for TE-35"
  N12:8  TE36_BIN  "Binary data for TE-36"
  N12:9  TE29_36_BTR_DATA9  "TE-29 thru TE-36 BTR Data 9"
  N12:9/0  TE29_UNDERRANGE
  N12:9/1  TE30_UNDERRANGE
  N12:9/2  TE31_UNDERRANGE
  N12:9/3  TE32_UNDERRANGE
  N12:9/4  TE33_UNDERRANGE
  N12:9/5  TE34_UNDERRANGE
  N12:9/6  TE35_UNDERRANGE
  N12:9/7  TE36_UNDERRANGE
  N12:9/8  TE29_OVERRANGE
  N12:9/9  TE30_OVERRANGE
  N12:9/10  TE31_OVERRANGE
  N12:9/11  TE32_OVERRANGE
  N12:9/12  TE33_OVERRANGE
  N12:9/13  TE34_OVERRANGE
  N12:9/14  TE35_OVERRANGE
  N12:9/15  TE36_OVERRANGE
  N12:10  TE29_36_BTR_DATA10  "TE-29 thru TE-36 BTR Data 10"
  N12:10/0  CJC_UNDERRANGE
  N12:10/1  CJC_OVERRANGE
  N12:10/2  BAD_STRUCTURE
  N12:10/3  DIAGNOSTIC_1_OF_3
  N12:10/4  DIAGNOSTIC_2_OF_3
  N12:10/5  DIAGNOSTIC_3_OF_3
  N12:10/6  NOT_USED1
  N12:10/8  CALIBRATION_RANGE
  N12:10/9  CALIBRATION_DONE
  N12:10/10  CALBRATION_BAD
  N12:28  MCC4_IE8_UNDERRANGE  "MCC RIO Slot 4 Under-Range Bits for all VFD Amps"
  N12:28/0  VFD01_AMP_UNDERRANGE  "VFD01 Amps Input Signal Broken or Under-Range"
  N12:28/1  VFD02_AMP_UNDERRANGE  "VFD02 Amps Input Signal Broken or Under-Range"
  N12:28/2  VFD03_AMP_UNDERRANGE  "VFD03 Amps Input Signal Broken or Under-Range"
  N12:28/3  VFD04_AMP_UNDERRANGE  "VFD04 Amps Input Signal Broken or Under-Range"
  N12:28/4  VFD05_AMP_UNDERRANGE  "VFD05 Amps Input Signal Broken or Under-Range"
  N12:28/5  VFD06_AMP_UNDERRANGE  "VFD06 Amps Input Signal Broken or Under-Range"
  N12:28/6  VFD07_AMP_UNDERRANGE  "VFD07 Amps Input Signal Broken or Under-Range"
  N12:28/7  VFD08_AMP_UNDERRANGE  "VFD08 Amps Input Signal Broken or Under-Range"
  N12:28/15  MCC4_IE8_CONFIG_ERR  "MCC RIO Slot 4 Unconfigured Error"
  N12:101  AI102_BIN_DATA
  N12:102  AI103_BIN_DATA
  N12:103  AI104_BIN_DATA
  N12:105  AI106_BIN_DATA
  N12:106  AI107_BIN_DATA
  N12:107  AI108_BIN_DATA
  N12:108  PN5_IE81_UNDERRANGE
  N12:111  AI110_BIN_DATA
  N12:112  AI111_BIN_DATA
  N12:113  AI112_BIN_DATA
  N12:114  AI113_BIN_DATA
  N12:115  AI114_BIN_DATA
  N12:116  AI115_BIN_DATA
  N12:117  AI116_BIN_DATA
  N12:118  PN5_IE82_UNDERRANGE
  N13:2  TE02_SETUP  "This File Determines Units (°C or °F) & Accuracy(0 or 0.0) for TE-2"
  N13:3  TE03_SETUP  "This File Determines Units (°C or °F) & Accuracy(0 or 0.0) for TE-3"
  N13:4  TE04_SETUP  "This File Determines Units (°C or °F) & Accuracy(0 or 0.0) for TE-4"
  N13:5  TE05_SETUP  "This File Determines Units (°C or °F) & Accuracy(0 or 0.0) for TE-5"
  N13:6  TE06_SETUP  "This File Determines Units (°C or °F) & Accuracy(0 or 0.0) for TE-6"
  N13:7  TE07_SETUP  "This File Determines Units (°C or °F) & Accuracy(0 or 0.0) for TE-7"
  N13:8  TE08_SETUP  "This File Determines Units (°C or °F) & Accuracy(0 or 0.0) for TE-8"
  N13:10  TE10_SETUP  "This File Determines Units (°C or °F) & Accuracy(0 or 0.0) for TE-10"
  N13:11  TE11_SETUP  "This File Determines Units (°C or °F) & Accuracy(0 or 0.0) for TE-11"
  N13:12  TE12_SETUP  "This File Determines Units (°C or °F) & Accuracy(0 or 0.0) for TE-12"
  N13:14  TE14_SETUP  "This File Determines Units (°C or °F) & Accuracy(0 or 0.0) for TE-14"
  N13:15  TE15_SETUP  "This File Determines Units (°C or °F) & Accuracy(0 or 0.0) for TE-15"
  N13:16  TE16_SETUP  "This File Determines Units (°C or °F) & Accuracy(0 or 0.0) for TE-16"
  N13:18  TE18_SETUP  "This File Determines Units (°C or °F) & Accuracy(0 or 0.0) for TE-18"
  N13:19  TE19_SETUP  "This File Determines Units (°C or °F) & Accuracy(0 or 0.0) for TE-19"
  N13:20  TE20_SETUP  "This File Determines Units (°C or °F) & Accuracy(0 or 0.0) for TE-20"
  N13:22  TE22_SETUP  "This File Determines Units (°C or °F) & Accuracy(0 or 0.0) for TE-22"
  N13:23  TE23_SETUP  "This File Determines Units (°C or °F) & Accuracy(0 or 0.0) for TE-23"
  N13:24  TE24_SETUP  "This File Determines Units (°C or °F) & Accuracy(0 or 0.0) for TE-24"
  N13:26  TE26_SETUP  "This File Determines Units (°C or °F) & Accuracy(0 or 0.0) for TE-26"
  N13:27  TE27_SETUP  "This File Determines Units (°C or °F) & Accuracy(0 or 0.0) for TE-27"
  N13:28  TE28_SETUP  "This File Determines Units (°C or °F) & Accuracy(0 or 0.0) for TE-28"
  N13:31  TE29_36_SETUP1  "RIO 1794-IT8 Setup Word 1 Set TE-29 thru TE-32 to Type "J" T/C's"
  N13:32  TE29_36_SETUP2  "RIO 1794-IT8 Setup Word 2 Set TE-31 thru TE-36 to Type "J" T/C's"
  N13:55  "Configure OE4 Output Type (4/20madc)"
  N13:121  AO102_BIN_OUTPUT  "AO-102 Rack 0, Slot 3 OE4, Channel 1 Binary Output Data"
  N13:122  AO103_BIN_OUTPUT  "AO-103 Rack 0, Slot 3 OE4, Channel 2 Binary Output Data"
  N13:123  AO104_BIN_OUTPUT  "AO-104 Rack 0, Slot 3 OE4, Channel 3 Binary Output Data"
  N13:125  "Configure OE4 Output Type (4/20madc)"
  N15:0/0  FIC211_TM  "FIC-21-1 Feed Flow No-1 PID Time Mode 0 = STI 1 = Timed"
  N15:0/2  FIC211_CM  "FIC-21-1 Feed Flow No-1 Control Mode 0 = Reverse (SP-PV) 1 = Direct (PV-SP)"
  N15:0/3  FIC211_OL  "FIC-21-1 Feed Flow No-1 Output Limiting Enabled"
  N15:0/4  FIC211_RG  "FIC-21-1 Feed Flow No-1 Reset/Gain Enhancement x 0.01 for both"
  N15:0/5  FIC211_SPS  "FIC-21-1 Feed Flow No-1 SetPoint Scaling Specified"
  N15:0/6  FIC211_TF  "FIC-21-1 Feed Flow No-1 1 = Loop Undate Time too Fast"
  N15:0/7  FIC211_DA  "FIC-21-1 Feed Flow No-1 Derivative Action 0 = On PV 1 = On Error"
  N15:0/8  FIC211_DBA  "FIC-21-1 Feed Flow No-1 1 = PV Within Deadband"
  N15:0/9  FIC211_UL  "FIC-21-1 Feed Flow No-1 Output Greaater Than Upper CV"
  N15:0/10  FIC211_LL  "FIC-21-1 Feed Flow No-1 Output Less Than Lower CV"
  N15:0/11  FIC211_SPA  "FIC-21-1 Feed Flow No-1 Setpoint Out of Range"
  N15:0/12  FIC211_PVA  "FIC-21-1 Feed Flow No-1 PV Out of Range"
  N15:0/13  FIC211_DN  "FIC-21-1 Feed Flow No-1 PID Done"
  N15:0/15  FIC211_EN  "FIC-21-1 Feed Flow No-1 PID Enabled"
  N15:1  FIC211_EC  "FIC-21-1 Feed Flow No-1 PID Sub Error Code"
  N15:3  FIC211_G  "FIC-21-1 Feed Flow No-1 Gain"
  N15:4  FIC211_TI  "FIC-21-1 Feed Flow No-1 Reset"
  N15:5  FIC211_TD  "FIC-21-1 Feed Flow No-1 Rate"
  N15:6  FIC211_FFD  "FIC-21-1 Feed Flow No-1 Feed Forward Bias"
  N15:9  FIC211_DB  "FIC-21-1 Feed Flow No-1 Deadband"
  N15:10  FIC211_C1  "FIC-21-1 Feed Flow No-1 Used by PID Statement Do Not Alter"
  N15:13  FIC211_TIM  "FIC-21-1 Feed Flow No-1 Last Loop Update Time"
  N15:15  FIC211_ERR  "FIC-21-1 Feed Flow No-1 Scaled Error"
  N15:16  FIC211_OUT  "FIC-21-1 Feed Flow No-1 Output 0/100%"
  N15:17  FIC211_C2  "FIC-21-1 Feed Flow No-1 Used by PID Statement Do Not Alter"
  N15:18  FIC211_C3  "FIC-21-1 Feed Flow No-1 Used by PID Statement Do Not Alter"
  N15:19  FIC211_C4  "FIC-21-1 Feed Flow No-1 Used by PID Statement Do Not Alter"
  N15:20  FIC211_C5  "FIC-21-1 Feed Flow No-1 Used by PID Statement Do Not Alter"
  N15:21  FIC211_C6  "FIC-21-1 Feed Flow No-1 Used by PID Statement Do Not Alter"
  N15:22  FIC211_C7  "FIC-21-1 Feed Flow No-1 Used by PID Statement Do Not Alter"
  N15:30/0  FIC212_TM  "FIC-21-2 Feed Flow No-2 PID Time Mode 0 = STI 1 = Timed"
  N15:30/2  FIC212_CM  "FIC-21-2 Feed Flow No-2 Control Mode 0 = Reverse (SP-PV) 1 = Direct (PV-SP)"
  N15:30/3  FIC212_OL  "FIC-21-2 Feed Flow No-2 Output Limiting Enabled"
  N15:30/4  FIC212_RG  "FIC-21-2 Feed Flow No-2 Reset/Gain Enhancement x 0.01 for both"
  N15:30/5  FIC212_SPS  "FIC-21-2 Feed Flow No-2 SetPoint Scaling Specified"
  N15:30/6  FIC212_TF  "FIC-21-2 Feed Flow No-2 1 = Loop Undate Time too Fast"
  N15:30/7  FIC212_DA  "FIC-21-2 Feed Flow No-2 Derivative Action 0 = On PV 1 = On Error"
  N15:30/8  FIC212_DBA  "FIC-21-2 Feed Flow No-2 1 = PV Within Deadband"
  N15:30/9  FIC212_UL  "FIC-21-2 Feed Flow No-2 Output Greaater Than Upper CV"
  N15:30/10  FIC212_LL  "FIC-21-2 Feed Flow No-2 Output Less Than Lower CV"
  N15:30/11  FIC212_SPA  "FIC-21-2 Feed Flow No-2 Setpoint Out of Range"
  N15:30/12  FIC212_PVA  "FIC-21-2 Feed Flow No-2 PV Out of Range"
  N15:30/13  FIC212_DN  "FIC-21-2 Feed Flow No-2 PID Done"
  N15:30/15  FIC212_EN  "FIC-21-2 Feed Flow No-2 PID Enabled"
  N15:31  FIC212_EC  "FIC-21-2 Feed Flow No-2 PID Sub Error Code"
  N15:33  FIC212_G  "FIC-21-2 Feed Flow No-2 Gain"
  N15:34  FIC212_TI  "FIC-21-2 Feed Flow No-2 Reset"
  N15:35  FIC212_TD  "FIC-21-2 Feed Flow No-2 Rate"
  N15:36  FIC212_FFD  "FIC-21-2 Feed Flow No-2 Feed Forward Bias"
  N15:39  FIC212_DB  "FIC-21-2 Feed Flow No-2 Deadband"
  N15:40  FIC212_C1  "FIC-21-2 Feed Flow No-2 Used by PID Statement Do Not Alter"
  N15:43  FIC212_TIM  "FIC-21-2 Feed Flow No-2 Last Loop Update Time"
  N15:45  FIC212_ERR  "FIC-21-2 Feed Flow No-2 Scaled Error"
  N15:46  FIC212_OUT  "FIC-21-2 Feed Flow No-2 Output 0/100%"
  N15:47  FIC212_C2  "FIC-21-2 Feed Flow No-2 Used by PID Statement Do Not Alter"
  N15:48  FIC212_C3  "FIC-21-2 Feed Flow No-2 Used by PID Statement Do Not Alter"
  N15:49  FIC212_C4  "FIC-21-2 Feed Flow No-2 Used by PID Statement Do Not Alter"
  N15:50  FIC212_C5  "FIC-21-2 Feed Flow No-2 Used by PID Statement Do Not Alter"
  N15:51  FIC212_C6  "FIC-21-2 Feed Flow No-2 Used by PID Statement Do Not Alter"
  N15:52  FIC212_C7  "FIC-21-2 Feed Flow No-2 Used by PID Statement Do Not Alter"
  N15:55  FIC212_OFF_OUTPUT  "FIC-21-2 Output When PUMP is Off"
  N15:60/0  PIC091_TM  "PIC-9-1 Vacuum Press No-1 PID Time Mode 0 = STI 1 = Timed"
  N15:60/2  PIC091_CM  "PIC-9-1 Vacuum Press No-1 Control Mode 0 = Reverse (SP-PV) 1 = Direct (PV-SP)"
  N15:60/3  PIC091_OL  "PIC-9-1 Vacuum Press No-1 Output Limiting Enabled"
  N15:60/4  PIC091_RG  "PIC-9-1 Vacuum Press No-1 Reset/Gain Enhancement x 0.01 for both"
  N15:60/5  PIC091_SPS  "PIC-9-1 Vacuum Press No-1 SetPoint Scaling Specified"
  N15:60/6  PIC091_TF  "PIC-9-1 Vacuum Press No-1 1 = Loop Undate Time too Fast"
  N15:60/7  PIC091_DA  "PIC-9-1 Vacuum Press No-1 Derivative Action 0 = On PV 1 = On Error"
  N15:60/8  PIC091_DBA  "PIC-9-1 Vacuum Press No-1 1 = PV Within Deadband"
  N15:60/9  PIC091_UL  "PIC-9-1 Vacuum Press No-1 Output Greaater Than Upper CV"
  N15:60/10  PIC091_LL  "PIC-9-1 Vacuum Press No-1 Output Less Than Lower CV"
  N15:60/11  PIC091_SPA  "PIC-9-1 Vacuum Press No-1 Setpoint Out of Range"
  N15:60/12  PIC091_PVA  "PIC-9-1 Vacuum Press No-1 PV Out of Range"
  N15:60/13  PIC091_DN  "PIC-9-1 Vacuum Press No-1 PID Done"
  N15:60/15  PIC091_EN  "PIC-9-1 Vacuum Press No-1 PID Enabled"
  N15:61  PIC091_EC  "PIC-9-1 Vacuum Press No-1 PID Sub Error Code"
  N15:63  PIC091_G  "PIC-9-1 Vacuum Press No-1 Gain"
  N15:64  PIC091_TI  "PIC-9-1 Vacuum Press No-1 Reset"
  N15:65  PIC091_TD  "PIC-9-1 Vacuum Press No-1 Rate"
  N15:66  PIC091_FFD  "PIC-9-1 Vacuum Press No-1 Feed Forward Bias"
  N15:69  PIC091_DB  "PIC-9-1 Vacuum Press No-1 Deadband"
  N15:70  PIC091_C1  "PIC-9-1 Vacuum Press No-1 Used by PID Statement Do Not Alter"
  N15:73  PIC091_TIM  "PIC-9-1 Vacuum Press No-1 Last Loop Update Time"
  N15:75  PIC091_ERR  "PIC-9-1 Vacuum Press No-1 Scaled Error"
  N15:76  PIC091_OUT  "PIC-9-1 Vacuum Press No-1 Output 0/100%"
  N15:77  PIC091_C2  "PIC-9-1 Vacuum Press No-1 Used by PID Statement Do Not Alter"
  N15:78  PIC091_C3  "PIC-9-1 Vacuum Press No-1 Used by PID Statement Do Not Alter"
  N15:79  PIC091_C4  "PIC-9-1 Vacuum Press No-1 Used by PID Statement Do Not Alter"
  N15:80  PIC091_C5  "PIC-9-1 Vacuum Press No-1 Used by PID Statement Do Not Alter"
  N15:81  PIC091_C6  "PIC-9-1 Vacuum Press No-1 Used by PID Statement Do Not Alter"
  N15:82  PIC091_C7  "PIC-9-1 Vacuum Press No-1 Used by PID Statement Do Not Alter"
  N15:90/0  PIC101_TM  "PIC-10-1 Vacuum Press No-2 PID Time Mode 0 = STI 1 = Timed"
  N15:90/2  PIC101_CM  "PIC-10-1 Vacuum Press No-2 Control Mode 0 = Reverse (SP-PV) 1 = Direct (PV-SP)"
  N15:90/3  PIC101_OL  "PIC-10-1 Vacuum Press No-2 Output Limiting Enabled"
  N15:90/4  PIC101_RG  "PIC-10-1 Vacuum Press No-2 Reset/Gain Enhancement x 0.01 for both"
  N15:90/5  PIC101_SPS  "PIC-10-1 Vacuum Press No-2 SetPoint Scaling Specified"
  N15:90/6  PIC101_TF  "PIC-10-1 Vacuum Press No-2 1 = Loop Undate Time too Fast"
  N15:90/7  PIC101_DA  "PIC-10-1 Vacuum Press No-2 Derivative Action 0 = On PV 1 = On Error"
  N15:90/8  PIC101_DBA  "PIC-10-1 Vacuum Press No-2 1 = PV Within Deadband"
  N15:90/9  PIC101_UL  "PIC-10-1 Vacuum Press No-2 Output Greaater Than Upper CV"
  N15:90/10  PIC101_LL  "PIC-10-1 Vacuum Press No-2 Output Less Than Lower CV"
  N15:90/11  PIC101_SPA  "PIC-10-1 Vacuum Press No-2 Setpoint Out of Range"
  N15:90/12  PIC101_PVA  "PIC-10-1 Vacuum Press No-2 PV Out of Range"
  N15:90/13  PIC101_DN  "PIC-10-1 Vacuum Press No-2 PID Done"
  N15:90/15  PIC101_EN  "PIC-10-1 Vacuum Press No-2 PID Enabled"
  N15:91  PIC101_EC  "PIC-10-1 Vacuum Press No-2 PID Sub Error Code"
  N15:93  PIC101_G  "PIC-10-1 Vacuum Press No-2 Gain"
  N15:94  PIC101_TI  "PIC-10-1 Vacuum Press No-2 Reset"
  N15:95  PIC101_TD  "PIC-10-1 Vacuum Press No-2 Rate"
  N15:96  PIC101_FFD  "PIC-10-1 Vacuum Press No-2 Feed Forward Bias"
  N15:99  PIC101_DB  "PIC-10-1 Vacuum Press No-2 Deadband"
  N15:100  PIC101_C1  "PIC-10-1 Vacuum Press No-2 Used by PID Statement Do Not Alter"
  N15:103  PIC101_TIM  "PIC-10-1 Vacuum Press No-2 Last Loop Update Time"
  N15:105  PIC101_ERR  "PIC-10-1 Vacuum Press No-2 Scaled Error"
  N15:106  PIC101_OUT  "PIC-10-1 Vacuum Press No-2 Output 0/100%"
  N15:107  PIC101_C2  "PIC-10-1 Vacuum Press No-2 Used by PID Statement Do Not Alter"
  N15:108  PIC101_C3  "PIC-10-1 Vacuum Press No-2 Used by PID Statement Do Not Alter"
  N15:109  PIC101_C4  "PIC-10-1 Vacuum Press No-2 Used by PID Statement Do Not Alter"
  N15:110  PIC101_C5  "PIC-10-1 Vacuum Press No-2 Used by PID Statement Do Not Alter"
  N15:111  PIC101_C6  "PIC-10-1 Vacuum Press No-2 Used by PID Statement Do Not Alter"
  N15:112  PIC101_C7  "PIC-10-1 Vacuum Press No-2 Used by PID Statement Do Not Alter"
  N15:150/0  PIC281_TM  "PIC-28-1 Steam Press PID Time Mode 0 = STI 1 = Timed"
  N15:150/2  PIC281_CM  "PIC-28-1 Steam Press Control Mode 0 = Reverse (SP-PV) 1 = Direct (PV-SP)"
  N15:150/3  PIC281_OL  "PIC-28-1 Steam Press Output Limiting Enabled"
  N15:150/4  PIC281_RG  "PIC-28-1 Steam Press Reset/Gain Enhancement x 0.01 for both"
  N15:150/5  PIC281_SPS  "PIC-28-1 Steam Press SetPoint Scaling Specified"
  N15:150/6  PIC281_TF  "PIC-28-1 Steam Press 1 = Loop Undate Time too Fast"
  N15:150/7  PIC281_DA  "PIC-28-1 Steam Press Derivative Action 0 = On PV 1 = On Error"
  N15:150/8  PIC281_DBA  "PIC-28-1 Steam Press 1 = PV Within Deadband"
  N15:150/9  PIC281_UL  "PIC-28-1 Steam Press Output Greaater Than Upper CV"
  N15:150/10  PIC281_LL  "PIC-28-1 Steam Press Output Less Than Lower CV"
  N15:150/11  PIC281_SPA  "PIC-28-1 Steam Press Setpoint Out of Range"
  N15:150/12  PIC281_PVA  "PIC-28-1 Steam Press PV Out of Range"
  N15:150/13  PIC281_DN  "PIC-28-1 Steam Press PID Done"
  N15:150/15  PIC281_EN  "PIC-28-1 Steam Press PID Enabled"
  N15:151  PIC281_EC  "PIC-28-1 Steam Press PID Sub Error Code"
  N15:153  PIC281_G  "PIC-28-1 Steam Press Gain"
  N15:154  PIC281_TI  "PIC-28-1 Steam Press Reset"
  N15:155  PIC281_TD  "PIC-28-1 Steam Press Rate"
  N15:156  PIC281_FFD  "PIC-28-1 Steam Press Feed Forward Bias"
  N15:159  PIC281_DB  "PIC-28-1 Steam Press Deadband"
  N15:160  PIC281_C1  "PIC-28-1 Steam Press Used by PID Statement Do Not Alter"
  N15:163  PIC281_TIM  "PIC-28-1 Steam Press Last Loop Update Time"
  N15:165  PIC281_ERR  "PIC-28-1 Steam Press Scaled Error"
  N15:166  PIC281_OUT  "PIC-28-1 Steam Press Output 0/100%"
  N15:167  PIC281_C2  "PIC-28-1 Steam Press Used by PID Statement Do Not Alter"
  N15:168  PIC281_C3  "PIC-28-1 Steam Press Used by PID Statement Do Not Alter"
  N15:169  PIC281_C4  "PIC-28-1 Steam Press Used by PID Statement Do Not Alter"
  N15:170  PIC281_C5  "PIC-28-1 Steam Press Used by PID Statement Do Not Alter"
  N15:171  PIC281_C6  "PIC-28-1 Steam Press Used by PID Statement Do Not Alter"
  N15:172  PIC281_C7  "PIC-28-1 Steam Press Used by PID Statement Do Not Alter"
  N15:180/0  PIC301_TM  "PIC-30-1 Water Press PID Time Mode 0 = STI 1 = Timed"
  N15:180/2  PIC301_CM  "PIC-30-1 Water Press Control Mode 0 = Reverse (SP-PV) 1 = Direct (PV-SP)"
  N15:180/3  PIC301_OL  "PIC-30-1 Water Press Output Limiting Enabled"
  N15:180/4  PIC301_RG  "PIC-30-1 Water Press Reset/Gain Enhancement x 0.01 for both"
  N15:180/5  PIC301_SPS  "PIC-30-1 Water Press SetPoint Scaling Specified"
  N15:180/6  PIC301_TF  "PIC-30-1 Water Press 1 = Loop Undate Time too Fast"
  N15:180/7  PIC301_DA  "PIC-30-1 Water Press Derivative Action 0 = On PV 1 = On Error"
  N15:180/8  PIC301_DBA  "PIC-30-1 Water Press 1 = PV Within Deadband"
  N15:180/9  PIC301_UL  "PIC-30-1 Water Press Output Greaater Than Upper CV"
  N15:180/10  PIC301_LL  "PIC-30-1 Water Press Output Less Than Lower CV"
  N15:180/11  PIC301_SPA  "PIC-30-1 Water Press Setpoint Out of Range"
  N15:180/12  PIC301_PVA  "PIC-30-1 Water Press PV Out of Range"
  N15:180/13  PIC301_DN  "PIC-30-1 Water Press PID Done"
  N15:180/15  PIC301_EN  "PIC-30-1 Water Press PID Enabled"
  N15:181  PIC301_EC  "PIC-30-1 Water Press PID Sub Error Code"
  N15:183  PIC301_G  "PIC-30-1 Water Press Gain"
  N15:184  PIC301_TI  "PIC-30-1 Water Press Reset"
  N15:185  PIC301_TD  "PIC-30-1 Water Press Rate"
  N15:186  PIC301_FFD  "PIC-30-1 Water Press Feed Forward Bias"
  N15:189  PIC301_DB  "PIC-30-1 Water Press Deadband"
  N15:190  PIC301_C1  "PIC-30-1 Water Press Used by PID Statement Do Not Alter"
  N15:191  PIC301_OMAX  "PIC-30-1 Water Press Output Maximum"
  N15:192  PIC301_OMIN  "PIC-30-1 Water Press Output Minimum"
  N15:193  PIC301_TIM  "PIC-30-1 Water Press Last Loop Update Time"
  N15:195  PIC301_ERR  "PIC-30-1 Water Press Scaled Error"
  N15:196  PIC301_OUT  "PIC-30-1 Water Press Output 0/100%"
  N15:197  PIC301_C2  "PIC-30-1 Water Press Used by PID Statement Do Not Alter"
  N15:198  PIC301_C3  "PIC-30-1 Water Press Used by PID Statement Do Not Alter"
  N15:199  PIC301_C4  "PIC-30-1 Water Press Used by PID Statement Do Not Alter"
  N15:200  PIC301_C5  "PIC-30-1 Water Press Used by PID Statement Do Not Alter"
  N15:201  PIC301_C6  "PIC-30-1 Water Press Used by PID Statement Do Not Alter"
  N15:202  PIC301_C7  "PIC-30-1 Water Press Used by PID Statement Do Not Alter"
  N16:0/0  FIC213_TM  "FIC-21-3 Feed Flow No-3 PID Time Mode 0 = STI 1 = Timed"
  N16:0/2  FIC213_CM  "FIC-21-3 Feed Flow No-3 Control Mode 0 = Reverse (SP-PV) 1 = Direct (PV-SP)"
  N16:0/3  FIC213_OL  "FIC-21-3 Feed Flow No-3 Output Limiting Enabled"
  N16:0/4  FIC213_RG  "FIC-21-3 Feed Flow No-3 Reset/Gain Enhancement x 0.01 for both"
  N16:0/5  FIC213_SPS  "FIC-21-3 Feed Flow No-3 SetPoint Scaling Specified"
  N16:0/6  FIC213_TF  "FIC-21-3 Feed Flow No-3 1 = Loop Undate Time too Fast"
  N16:0/7  FIC213_DA  "FIC-21-3 Feed Flow No-3 Derivative Action 0 = On PV 1 = On Error"
  N16:0/8  FIC213_DBA  "FIC-21-3 Feed Flow No-3 1 = PV Within Deadband"
  N16:0/9  FIC213_UL  "FIC-21-3 Feed Flow No-3 Output Greaater Than Upper CV"
  N16:0/10  FIC213_LL  "FIC-21-3 Feed Flow No-3 Output Less Than Lower CV"
  N16:0/11  FIC213_SPA  "FIC-21-3 Feed Flow No-3 Setpoint Out of Range"
  N16:0/12  FIC213_PVA  "FIC-21-3 Feed Flow No-3 PV Out of Range"
  N16:0/13  FIC213_DN  "FIC-21-3 Feed Flow No-3 PID Done"
  N16:0/15  FIC213_EN  "FIC-21-3 Feed Flow No-3 PID Enabled"
  N16:1  FIC213_EC  "FIC-21-3 Feed Flow No-3 PID Sub Error Code"
  N16:3  FIC213_G  "FIC-21-3 Feed Flow No-3 Gain"
  N16:4  FIC213_TI  "FIC-21-3 Feed Flow No-3 Reset"
  N16:5  FIC213_TD  "FIC-21-3 Feed Flow No-3 Rate"
  N16:6  FIC213_FFD  "FIC-21-3 Feed Flow No-3 Feed Forward Bias"
  N16:9  FIC213_DB  "FIC-21-3 Feed Flow No-3 Deadband"
  N16:10  FIC213_C1  "FIC-21-3 Feed Flow No-3 Used by PID Statement Do Not Alter"
  N16:13  FIC213_TIM  "FIC-21-3 Feed Flow No-3 Last Loop Update Time"
  N16:15  FIC213_ERR  "FIC-21-3 Feed Flow No-3 Scaled Error"
  N16:16  FIC213_OUT  "FIC-21-3 Feed Flow No-3 Output 0/100%"
  N16:17  FIC213_C2  "FIC-21-3 Feed Flow No-3 Used by PID Statement Do Not Alter"
  N16:18  FIC213_C3  "FIC-21-3 Feed Flow No-3 Used by PID Statement Do Not Alter"
  N16:19  FIC213_C4  "FIC-21-3 Feed Flow No-3 Used by PID Statement Do Not Alter"
  N16:20  FIC213_C5  "FIC-21-3 Feed Flow No-3 Used by PID Statement Do Not Alter"
  N16:21  FIC213_C6  "FIC-21-3 Feed Flow No-3 Used by PID Statement Do Not Alter"
  N16:22  FIC213_C7  "FIC-21-3 Feed Flow No-3 Used by PID Statement Do Not Alter"
  N16:25  FIC213_OFF_OUTPUT  "FIC-21-3 Output When PUMP is Off"
  N16:30/0  FIC214_TM  "FIC-21-4 Feed Flow No-4 PID Time Mode 0 = STI 1 = Timed"
  N16:30/2  FIC214_CM  "FIC-21-4 Feed Flow No-4 Control Mode 0 = Reverse (SP-PV) 1 = Direct (PV-SP)"
  N16:30/3  FIC214_OL  "FIC-21-4 Feed Flow No-4 Output Limiting Enabled"
  N16:30/4  FIC214_RG  "FIC-21-4 Feed Flow No-4 Reset/Gain Enhancement x 0.01 for both"
  N16:30/5  FIC214_SPS  "FIC-21-4 Feed Flow No-4 SetPoint Scaling Specified"
  N16:30/6  FIC214_TF  "FIC-21-4 Feed Flow No-4 1 = Loop Undate Time too Fast"
  N16:30/7  FIC214_DA  "FIC-21-4 Feed Flow No-4 Derivative Action 0 = On PV 1 = On Error"
  N16:30/8  FIC214_DBA  "FIC-21-4 Feed Flow No-4 1 = PV Within Deadband"
  N16:30/9  FIC214_UL  "FIC-21-4 Feed Flow No-4 Output Greaater Than Upper CV"
  N16:30/10  FIC214_LL  "FIC-21-4 Feed Flow No-4 Output Less Than Lower CV"
  N16:30/11  FIC214_SPA  "FIC-21-4 Feed Flow No-4 Setpoint Out of Range"
  N16:30/12  FIC214_PVA  "FIC-21-4 Feed Flow No-4 PV Out of Range"
  N16:30/13  FIC214_DN  "FIC-21-4 Feed Flow No-4 PID Done"
  N16:30/15  FIC214_EN  "FIC-21-4 Feed Flow No-4 PID Enabled"
  N16:31  FIC214_EC  "FIC-21-4 Feed Flow No-4 PID Sub Error Code"
  N16:33  FIC214_G  "FIC-21-4 Feed Flow No-4 Gain"
  N16:34  FIC214_TI  "FIC-21-4 Feed Flow No-4 Reset"
  N16:35  FIC214_TD  "FIC-21-4 Feed Flow No-4 Rate"
  N16:36  FIC214_FFD  "FIC-21-4 Feed Flow No-4 Feed Forward Bias"
  N16:39  FIC214_DB  "FIC-21-4 Feed Flow No-4 Deadband"
  N16:40  FIC214_C1  "FIC-21-4 Feed Flow No-4 Used by PID Statement Do Not Alter"
  N16:43  FIC214_TIM  "FIC-21-4 Feed Flow No-4 Last Loop Update Time"
  N16:45  FIC214_ERR  "FIC-21-4 Feed Flow No-4 Scaled Error"
  N16:46  FIC214_OUT  "FIC-21-4 Feed Flow No-4 Output 0/100%"
  N16:47  FIC214_C2  "FIC-21-4 Feed Flow No-4 Used by PID Statement Do Not Alter"
  N16:48  FIC214_C3  "FIC-21-4 Feed Flow No-4 Used by PID Statement Do Not Alter"
  N16:49  FIC214_C4  "FIC-21-4 Feed Flow No-4 Used by PID Statement Do Not Alter"
  N16:50  FIC214_C5  "FIC-21-4 Feed Flow No-4 Used by PID Statement Do Not Alter"
  N16:51  FIC214_C6  "FIC-21-4 Feed Flow No-4 Used by PID Statement Do Not Alter"
  N16:52  FIC214_C7  "FIC-21-4 Feed Flow No-4 Used by PID Statement Do Not Alter"
  N16:55  FIC214_OFF_OUTPUT  "FIC-21-4 Output When PUMP is Off"
  N16:60/0  PIC461_TM  "PIC-46-1 Flash Evap Feed Pres PID Time Mode 0 = STI 1 = Timed"
  N16:60/2  PIC461_CM  "PIC-46-1 Flash Evap Feed Pres Control Mode 0 = Reverse (SP-PV) 1 = Direct (PV-SP)"
  N16:60/3  PIC461_OL  "PIC-46-1 Flash Evap Feed Pres Output Limiting Enabled"
  N16:60/4  PIC461_RG  "PIC-46-1 Flash Evap Feed Pres Reset/Gain Enhancement x 0.01 for both"
  N16:60/5  PIC461_SPS  "PIC-46-1 Flash Evap Feed Pres SetPoint Scaling Specified"
  N16:60/6  PIC461_TF  "PIC-46-1 Flash Evap Feed Pres 1 = Loop Undate Time too Fast"
  N16:60/7  PIC461_DA  "PIC-46-1 Flash Evap Feed Pres Derivative Action 0 = On PV 1 = On Error"
  N16:60/8  PIC461_DBA  "PIC-46-1 Flash Evap Feed Pres 1 = PV Within Deadband"
  N16:60/9  PIC461_UL  "PIC-46-1 Flash Evap Feed Pres Output Greaater Than Upper CV"
  N16:60/10  PIC461_LL  "PIC-46-1 Flash Evap Feed Pres Output Less Than Lower CV"
  N16:60/11  PIC461_SPA  "PIC-46-1 Flash Evap Feed Pres Setpoint Out of Range"
  N16:60/12  PIC461_PVA  "PIC-46-1 Flash Evap Feed Pres PV Out of Range"
  N16:60/13  PIC461_DN  "PIC-46-1 Flash Evap Feed Pres PID Done"
  N16:60/15  PIC461_EN  "PIC-46-1 Flash Evap Feed Pres PID Enabled"
  N16:61  PIC461_EC  "PIC-46-1 Flash Evap Feed Pres PID Sub Error Code"
  N16:63  PIC461_G  "PIC-46-1 Flash Evap Feed Pres Gain"
  N16:64  PIC461_TI  "PIC-46-1 Flash Evap Feed Pres Reset"
  N16:65  PIC461_TD  "PIC-46-1 Flash Evap Feed Pres Rate"
  N16:66  PIC461_FFD  "PIC-46-1 Flash Evap Feed Pres Feed Forward Bias"
  N16:69  PIC461_DB  "PIC-46-1 Flash Evap Feed Pres Deadband"
  N16:70  PIC461_C1  "PIC-46-1 Flash Evap Feed Pres Used by PID Statement Do Not Alter"
  N16:73  PIC461_TIM  "PIC-46-1 Flash Evap Feed Pres Last Loop Update Time"
  N16:75  PIC461_ERR  "PIC-46-1 Flash Evap Feed Pres Scaled Error"
  N16:76  PIC461_OUT  "PIC-46-1 Flash Evap Feed Pres Output 0/100%"
  N16:77  PIC461_C2  "PIC-46-1 Flash Evap Feed Pres Used by PID Statement Do Not Alter"
  N16:78  PIC461_C3  "PIC-46-1 Flash Evap Feed Pres Used by PID Statement Do Not Alter"
  N16:79  PIC461_C4  "PIC-46-1 Flash Evap Feed Pres Used by PID Statement Do Not Alter"
  N16:80  PIC461_C5  "PIC-46-1 Flash Evap Feed Pres Used by PID Statement Do Not Alter"
  N16:81  PIC461_C6  "PIC-46-1 Flash Evap Feed Pres Used by PID Statement Do Not Alter"
  N16:82  PIC461_C7  "PIC-46-1 Flash Evap Feed Pres Used by PID Statement Do Not Alter"
  N16:85  PIC461_OFF_OUTPUT  "PIC-46-1 Output When PUMP is Off"
  N16:150/0  LIC221_TM  "LIC-22-1 Level No-1 PID Time Mode 0 = STI 1 = Timed"
  N16:150/2  LIC221_CM  "LIC-22-1 Level No-1 Control Mode 0 = Reverse (SP-PV) 1 = Direct (PV-SP)"
  N16:150/3  LIC221_OL  "LIC-22-1 Level No-1 Output Limiting Enabled"
  N16:150/4  LIC221_RG  "LIC-22-1 Level No-1 Reset/Gain Enhancement x 0.01 for both"
  N16:150/5  LIC221_SPS  "LIC-22-1 Level No-1 SetPoint Scaling Specified"
  N16:150/6  LIC221_TF  "LIC-22-1 Level No-1 1 = Loop Undate Time too Fast"
  N16:150/7  LIC221_DA  "LIC-22-1 Level No-1 Derivative Action 0 = On PV 1 = On Error"
  N16:150/8  LIC221_DBA  "LIC-22-1 Level No-1 1 = PV Within Deadband"
  N16:150/9  LIC221_UL  "LIC-22-1 Level No-1 Output Greaater Than Upper CV"
  N16:150/10  LIC221_LL  "LIC-22-1 Level No-1 Output Less Than Lower CV"
  N16:150/11  LIC221_SPA  "LIC-22-1 Level No-1 Setpoint Out of Range"
  N16:150/12  LIC221_PVA  "LIC-22-1 Level No-1 PV Out of Range"
  N16:150/13  LIC221_DN  "LIC-22-1 Level No-1 PID Done"
  N16:150/15  LIC221_EN  "LIC-22-1 Level No-1 PID Enabled"
  N16:151  LIC221_EC  "LIC-22-1 Level No-1 PID Sub Error Code"
  N16:153  LIC221_G  "LIC-22-1 Level No-1 Gain"
  N16:154  LIC221_TI  "LIC-22-1 Level No-1 Reset"
  N16:155  LIC221_TD  "LIC-22-1 Level No-1 Rate"
  N16:156  LIC221_FFD  "LIC-22-1 Level No-1 Feed Forward Bias"
  N16:159  LIC221_DB  "LIC-22-1 Level No-1 Deadband"
  N16:160  LIC221_C1  "LIC-22-1 Level No-1 Used by PID Statement Do Not Alter"
  N16:163  LIC221_TIM  "LIC-22-1 Level No-1 Last Loop Update Time"
  N16:165  LIC221_ERR  "LIC-22-1 Level No-1 Scaled Error"
  N16:166  LIC221_OUT  "LIC-22-1 Level No-1 Output 0/100%"
  N16:167  LIC221_C2  "LIC-22-1 Level No-1 Used by PID Statement Do Not Alter"
  N16:168  LIC221_C3  "LIC-22-1 Level No-1 Used by PID Statement Do Not Alter"
  N16:169  LIC221_C4  "LIC-22-1 Level No-1 Used by PID Statement Do Not Alter"
  N16:170  LIC221_C5  "LIC-22-1 Level No-1 Used by PID Statement Do Not Alter"
  N16:171  LIC221_C6  "LIC-22-1 Level No-1 Used by PID Statement Do Not Alter"
  N16:172  LIC221_C7  "LIC-22-1 Level No-1 Used by PID Statement Do Not Alter"
  N16:175  LIC221_OFF_OUTPUT  "LIC-22-1 Output When PUMP is Off"
  N17:0/0  TIC111_TM  "TIC-11-1 Tempered Water No-1 PID Time Mode 0 = STI 1 = Timed"
  N17:0/2  TIC111_CM  "TIC-11-1 Tempered Water No-1 Control Mode 0 = Reverse (SP-PV) 1 = Direct (PV-SP)"
  N17:0/3  TIC111_OL  "TIC-11-1 Tempered Water No-1 Output Limiting Enabled"
  N17:0/4  TIC111_RG  "TIC-11-1 Tempered Water No-1 Reset/Gain Enhancement x 0.01 for both"
  N17:0/5  TIC111_SPS  "TIC-11-1 Tempered Water No-1 SetPoint Scaling Specified"
  N17:0/6  TIC111_TF  "TIC-11-1 Tempered Water No-1 1 = Loop Undate Time too Fast"
  N17:0/7  TIC111_DA  "TIC-11-1 Tempered Water No-1 Derivative Action 0 = On PV 1 = On Error"
  N17:0/8  TIC111_DBA  "TIC-11-1 Tempered Water No-1 1 = PV Within Deadband"
  N17:0/9  TIC111_UL  "TIC-11-1 Tempered Water No-1 Output Greaater Than Upper CV"
  N17:0/10  TIC111_LL  "TIC-11-1 Tempered Water No-1 Output Less Than Lower CV"
  N17:0/11  TIC111_SPA  "TIC-11-1 Tempered Water No-1 Setpoint Out of Range"
  N17:0/12  TIC111_PVA  "TIC-11-1 Tempered Water No-1 PV Out of Range"
  N17:0/13  TIC111_DN  "TIC-11-1 Tempered Water No-1 PID Done"
  N17:0/15  TIC111_EN  "TIC-11-1 Tempered Water No-1 PID Enabled"
  N17:1  TIC111_EC  "TIC-11-1 Tempered Water No-1 PID Sub Error Code"
  N17:3  TIC111_G  "TIC-11-1 Tempered Water No-1 Gain"
  N17:4  TIC111_TI  "TIC-11-1 Tempered Water No-1 Reset"
  N17:5  TIC111_TD  "TIC-11-1 Tempered Water No-1 Rate"
  N17:6  TIC111_FFD  "TIC-11-1 Tempered Water No-1 Feed Forward Bias"
  N17:9  TIC111_DB  "TIC-11-1 Tempered Water No-1 Deadband"
  N17:10  TIC111_C1  "TIC-11-1 Tempered Water No-1 Used by PID Statement Do Not Alter"
  N17:11  TIC111_OMAX  "TIC-11-1 Tempered Water No-1 Output Maximum"
  N17:12  TIC111_OMIN  "TIC-11-1 Tempered Water No-1 Output Minimum"
  N17:13  TIC111_TIM  "TIC-11-1 Tempered Water No-1 Last Loop Update Time"
  N17:15  TIC111_ERR  "TIC-11-1 Tempered Water No-1 Scaled Error"
  N17:16  TIC111_OUT  "TIC-11-1 Tempered Water No-1 Output 0/100%"
  N17:17  TIC111_C2  "TIC-11-1 Tempered Water No-1 Used by PID Statement Do Not Alter"
  N17:18  TIC111_C3  "TIC-11-1 Tempered Water No-1 Used by PID Statement Do Not Alter"
  N17:19  TIC111_C4  "TIC-11-1 Tempered Water No-1 Used by PID Statement Do Not Alter"
  N17:20  TIC111_C5  "TIC-11-1 Tempered Water No-1 Used by PID Statement Do Not Alter"
  N17:21  TIC111_C6  "TIC-11-1 Tempered Water No-1 Used by PID Statement Do Not Alter"
  N17:22  TIC111_C7  "TIC-11-1 Tempered Water No-1 Used by PID Statement Do Not Alter"
  N17:30/0  TIC121_TM  "TIC-12-1 Tempered Water No-2 PID Time Mode 0 = STI 1 = Timed"
  N17:30/3  TIC121_OL  "TIC-12-1 Tempered Water No-2 Output Limiting Enabled"
  N17:30/4  TIC121_RG  "TIC-12-1 Tempered Water No-2 Reset/Gain Enhancement x 0.01 for both"
  N17:30/5  TIC121_SPS  "TIC-12-1 Tempered Water No-2 SetPoint Scaling Specified"
  N17:30/6  TIC121_TF  "TIC-12-1 Tempered Water No-2 1 = Loop Undate Time too Fast"
  N17:30/7  TIC121_DA  "TIC-12-1 Tempered Water No-2 Derivative Action 0 = On PV 1 = On Error"
  N17:30/8  TIC121_DBA  "TIC-12-1 Tempered Water No-2 1 = PV Within Deadband"
  N17:30/9  TIC121_UL  "TIC-12-1 Tempered Water No-2 Output Greaater Than Upper CV"
  N17:30/10  TIC121_LL  "TIC-12-1 Tempered Water No-2 Output Less Than Lower CV"
  N17:30/11  TIC121_SPA  "TIC-12-1 Tempered Water No-2 Setpoint Out of Range"
  N17:30/12  TIC121_PVA  "TIC-12-1 Tempered Water No-2 PV Out of Range"
  N17:30/13  TIC121_DN  "TIC-12-1 Tempered Water No-2 PID Done"
  N17:30/15  TIC121_EN  "TIC-12-1 Tempered Water No-2 PID Enabled"
  N17:31  TIC121_EC  "TIC-12-1 Tempered Water No-2 PID Sub Error Code"
  N17:33  TIC121_G  "TIC-12-1 Tempered Water No-2 Gain"
  N17:34  TIC121_TI  "TIC-12-1 Tempered Water No-2 Reset"
  N17:35  TIC121_TD  "TIC-12-1 Tempered Water No-2 Rate"
  N17:36  TIC121_FFD  "TIC-12-1 Tempered Water No-2 Feed Forward Bias"
  N17:39  TIC121_DB  "TIC-12-1 Tempered Water No-2 Deadband"
  N17:40  TIC121_C1  "TIC-12-1 Tempered Water No-2 Used by PID Statement Do Not Alter"
  N17:41  TIC121_OMAX  "TIC-12-1 Tempered Water No-2 Output Maximum"
  N17:42  TIC121_OMIN  "TIC-12-1 Tempered Water No-2 Output Minimum"
  N17:43  TIC121_TIM  "TIC-12-1 Tempered Water No-2 Last Loop Update Time"
  N17:45  TIC121_ERR  "TIC-12-1 Tempered Water No-2 Scaled Error"
  N17:46  TIC121_OUT  "TIC-12-1 Tempered Water No-2 Output 0/100%"
  N17:47  TIC121_C2  "TIC-12-1 Tempered Water No-2 Used by PID Statement Do Not Alter"
  N17:48  TIC121_C3  "TIC-12-1 Tempered Water No-2 Used by PID Statement Do Not Alter"
  N17:49  TIC121_C4  "TIC-12-1 Tempered Water No-2 Used by PID Statement Do Not Alter"
  N17:50  TIC121_C5  "TIC-12-1 Tempered Water No-2 Used by PID Statement Do Not Alter"
  N17:51  TIC121_C6  "TIC-12-1 Tempered Water No-2 Used by PID Statement Do Not Alter"
  N17:52  TIC121_C7  "TIC-12-1 Tempered Water No-2 Used by PID Statement Do Not Alter"
  N17:60/0  TIC151_TM  "TIC-15-1 Tempered Oil No-1 PID Time Mode 0 = STI 1 = Timed"
  N17:60/2  TIC151_CM  "TIC-15-1 Tempered Oil No-1 Control Mode 0 = Reverse (SP-PV) 1 = Direct (PV-SP)"
  N17:60/3  TIC151_OL  "TIC-15-1 Tempered Oil No-1 Output Limiting Enabled"
  N17:60/4  TIC151_RG  "TIC-15-1 Tempered Oil No-1 Reset/Gain Enhancement x 0.01 for both"
  N17:60/5  TIC151_SPS  "TIC-15-1 Tempered Oil No-1 SetPoint Scaling Specified"
  N17:60/6  TIC151_TF  "TIC-15-1 Tempered Oil No-1 1 = Loop Undate Time too Fast"
  N17:60/7  TIC151_DA  "TIC-15-1 Tempered Oil No-1 Derivative Action 0 = On PV 1 = On Error"
  N17:60/8  TIC151_DBA  "TIC-15-1 Tempered Oil No-1 1 = PV Within Deadband"
  N17:60/9  TIC151_UL  "TIC-15-1 Tempered Oil No-1 Output Greaater Than Upper CV"
  N17:60/10  TIC151_LL  "TIC-15-1 Tempered Oil No-1 Output Less Than Lower CV"
  N17:60/11  TIC151_SPA  "TIC-15-1 Tempered Oil No-1 Setpoint Out of Range"
  N17:60/12  TIC151_PVA  "TIC-15-1 Tempered Oil No-1 PV Out of Range"
  N17:60/13  TIC151_DN  "TIC-15-1 Tempered Oil No-1 PID Done"
  N17:60/15  TIC151_EN  "TIC-15-1 Tempered Oil No-1 PID Enabled"
  N17:61  TIC151_EC  "TIC-15-1 Tempered Oil No-1 PID Sub Error Code"
  N17:63  TIC151_G  "TIC-15-1 Tempered Oil No-1 Gain"
  N17:64  TIC151_TI  "TIC-15-1 Tempered Oil No-1 Reset"
  N17:65  TIC151_TD  "TIC-15-1 Tempered Oil No-1 Rate"
  N17:66  TIC151_FFD  "TIC-15-1 Tempered Oil No-1 Feed Forward Bias"
  N17:69  TIC151_DB  "TIC-15-1 Tempered Oil No-1 Deadband"
  N17:70  TIC151_C1  "TIC-15-1 Tempered Oil No-1 Used by PID Statement Do Not Alter"
  N17:71  TIC151_OMAX  "TIC-15-1 Tempered Oil No-1 Output Maximum"
  N17:72  TIC151_OMIN  "TIC-15-1 Tempered Oil No-1 Output Minimum"
  N17:73  TIC151_TIM  "TIC-15-1 Tempered Oil No-1 Last Loop Update Time"
  N17:75  TIC151_ERR  "TIC-15-1 Tempered Oil No-1 Scaled Error"
  N17:76  TIC151_OUT  "TIC-15-1 Tempered Oil No-1 Output 0/100%"
  N17:77  TIC151_C2  "TIC-15-1 Tempered Oil No-1 Used by PID Statement Do Not Alter"
  N17:78  TIC151_C3  "TIC-15-1 Tempered Oil No-1 Used by PID Statement Do Not Alter"
  N17:79  TIC151_C4  "TIC-15-1 Tempered Oil No-1 Used by PID Statement Do Not Alter"
  N17:80  TIC151_C5  "TIC-15-1 Tempered Oil No-1 Used by PID Statement Do Not Alter"
  N17:81  TIC151_C6  "TIC-15-1 Tempered Oil No-1 Used by PID Statement Do Not Alter"
  N17:82  TIC151_C7  "TIC-15-1 Tempered Oil No-1 Used by PID Statement Do Not Alter"
  N17:90/0  TIC241_TM  "TIC-24-1 Hot Oil Temp PID Time Mode 0 = STI 1 = Timed"
  N17:90/2  TIC241_CM  "TIC-24-1 Hot Oil Temp Control Mode 0 = Reverse (SP-PV) 1 = Direct (PV-SP)"
  N17:90/3  TIC241_OL  "TIC-24-1 Hot Oil Temp Output Limiting Enabled"
  N17:90/4  TIC241_RG  "TIC-24-1 Hot Oil Temp Reset/Gain Enhancement x 0.01 for both"
  N17:90/5  TIC241_SPS  "TIC-24-1 Hot Oil Temp SetPoint Scaling Specified"
  N17:90/6  TIC241_TF  "TIC-24-1 Hot Oil Temp 1 = Loop Undate Time too Fast"
  N17:90/7  TIC241_DA  "TIC-24-1 Hot Oil Temp Derivative Action 0 = On PV 1 = On Error"
  N17:90/8  TIC241_DBA  "TIC-24-1 Hot Oil Temp 1 = PV Within Deadband"
  N17:90/9  TIC241_UL  "TIC-24-1 Hot Oil Temp Output Greaater Than Upper CV"
  N17:90/10  TIC241_LL  "TIC-24-1 Hot Oil Temp Output Less Than Lower CV"
  N17:90/11  TIC241_SPA  "TIC-24-1 Hot Oil Temp Setpoint Out of Range"
  N17:90/12  TIC241_PVA  "TIC-24-1 Hot Oil Temp PV Out of Range"
  N17:90/13  TIC241_DN  "TIC-24-1 Hot Oil Temp PID Done"
  N17:90/15  TIC241_EN  "TIC-24-1 Hot Oil Temp PID Enabled"
  N17:91  TIC241_EC  "TIC-24-1 Hot Oil Temp PID Sub Error Code"
  N17:93  TIC241_G  "TIC-24-1 Hot Oil Temp Gain"
  N17:94  TIC241_TI  "TIC-24-1 Hot Oil Temp Reset"
  N17:95  TIC241_TD  "TIC-24-1 Hot Oil Temp Rate"
  N17:96  TIC241_FFD  "TIC-24-1 Hot Oil Temp Feed Forward Bias"
  N17:99  TIC241_DB  "TIC-24-1 Hot Oil Temp Deadband"
  N17:100  TIC241_C1  "TIC-24-1 Hot Oil Temp Used by PID Statement Do Not Alter"
  N17:102  TIC241_OMIN  "TIC-24-1 Hot Oil Temp Output Minimum"
  N17:103  TIC241_TIM  "TIC-24-1 Hot Oil Temp Last Loop Update Time"
  N17:105  TIC241_ERR  "TIC-24-1 Hot Oil Temp Scaled Error"
  N17:106  TIC241_OUT  "TIC-24-1 Hot Oil Temp Output 0/100%"
  N17:107  TIC241_C2  "TIC-24-1 Hot Oil Temp Used by PID Statement Do Not Alter"
  N17:108  TIC241_C3  "TIC-24-1 Hot Oil Temp Used by PID Statement Do Not Alter"
  N17:109  TIC241_C4  "TIC-24-1 Hot Oil Temp Used by PID Statement Do Not Alter"
  N17:110  TIC241_C5  "TIC-24-1 Hot Oil Temp Used by PID Statement Do Not Alter"
  N17:111  TIC241_C6  "TIC-24-1 Hot Oil Temp Used by PID Statement Do Not Alter"
  N17:112  TIC241_C7  "TIC-24-1 Hot Oil Temp Used by PID Statement Do Not Alter"
  N17:120/0  TIC371_TM  "TIC-37-1 Tempered Oil No-3 PID Time Mode 0 = STI 1 = Timed"
  N17:120/2  TIC371_CM  "TIC-37-1 Tempered Oil No-3 Control Mode 0 = Reverse (SP-PV) 1 = Direct (PV-SP)"
  N17:120/3  TIC371_OL  "TIC-37-1 Tempered Oil No-3 Output Limiting Enabled"
  N17:120/4  TIC371_RG  "TIC-37-1 Tempered Oil No-3 Reset/Gain Enhancement x 0.01 for both"
  N17:120/5  TIC371_SPS  "TIC-37-1 Tempered Oil No-3 SetPoint Scaling Specified"
  N17:120/6  TIC371_TF  "TIC-37-1 Tempered Oil No-3 1 = Loop Undate Time too Fast"
  N17:120/7  TIC371_DA  "TIC-37-1 Tempered Oil No-3 Derivative Action 0 = On PV 1 = On Error"
  N17:120/8  TIC371_DBA  "TIC-37-1 Tempered Oil No-3 1 = PV Within Deadband"
  N17:120/9  TIC371_UL  "TIC-37-1 Tempered Oil No-3 Output Greaater Than Upper CV"
  N17:120/10  TIC371_LL  "TIC-37-1 Tempered Oil No-3 Output Less Than Lower CV"
  N17:120/11  TIC371_SPA  "TIC-37-1 Tempered Oil No-3 Setpoint Out of Range"
  N17:120/12  TIC371_PVA  "TIC-37-1 Tempered Oil No-3 PV Out of Range"
  N17:120/13  TIC371_DN  "TIC-37-1 Tempered Oil No-3 PID Done"
  N17:120/15  TIC371_EN  "TIC-37-1 Tempered Oil No-3 PID Enabled"
  N17:121  TIC371_EC  "TIC-37-1 Tempered Oil No-3 PID Sub Error Code"
  N17:123  TIC371_G  "TIC-37-1 Tempered Oil No-3 Gain"
  N17:124  TIC371_TI  "TIC-37-1 Tempered Oil No-3 Reset"
  N17:125  TIC371_TD  "TIC-37-1 Tempered Oil No-3 Rate"
  N17:126  TIC371_FFD  "TIC-37-1 Tempered Oil No-3 Feed Forward Bias"
  N17:129  TIC371_DB  "TIC-37-1 Tempered Oil No-3 Deadband"
  N17:130  TIC371_C1  "TIC-37-1 Tempered Oil No-3 Used by PID Statement Do Not Alter"
  N17:131  TIC371_OMAX  "TIC-37-1 Tempered Oil No-3 Output Maximum"
  N17:132  TIC371_OMIN  "TIC-37-1 Tempered Oil No-3 Output Minimum"
  N17:133  TIC371_TIM  "TIC-37-1 Tempered Oil No-3 Last Loop Update Time"
  N17:135  TIC371_ERR  "TIC-37-1 Tempered Oil No-3 Scaled Error"
  N17:136  TIC371_OUT  "TIC-37-1 Tempered Oil No-3 Output 0/100%"
  N17:137  TIC371_C2  "TIC-37-1 Tempered Oil No-3 Used by PID Statement Do Not Alter"
  N17:138  TIC371_C3  "TIC-37-1 Tempered Oil No-3 Used by PID Statement Do Not Alter"
  N17:139  TIC371_C4  "TIC-37-1 Tempered Oil No-3 Used by PID Statement Do Not Alter"
  N17:140  TIC371_C5  "TIC-37-1 Tempered Oil No-3 Used by PID Statement Do Not Alter"
  N17:141  TIC371_C6  "TIC-37-1 Tempered Oil No-3 Used by PID Statement Do Not Alter"
  N17:142  TIC371_C7  "TIC-37-1 Tempered Oil No-3 Used by PID Statement Do Not Alter"
  N17:150/0  TIC401_TM  "TIC-40-1 Tempered Oil No-2 PID Time Mode 0 = STI 1 = Timed"
  N17:150/2  TIC401_CM  "TIC-40-1 Tempered Oil No-2 Control Mode 0 = Reverse (SP-PV) 1 = Direct (PV-SP)"
  N17:150/3  TIC401_OL  "TIC-40-1 Tempered Oil No-2 Output Limiting Enabled"
  N17:150/4  TIC401_RG  "TIC-40-1 Tempered Oil No-2 Reset/Gain Enhancement x 0.01 for both"
  N17:150/5  TIC401_SPS  "TIC-40-1 Tempered Oil No-2 SetPoint Scaling Specified"
  N17:150/6  TIC401_TF  "TIC-40-1 Tempered Oil No-2 1 = Loop Undate Time too Fast"
  N17:150/7  TIC401_DA  "TIC-40-1 Tempered Oil No-2 Derivative Action 0 = On PV 1 = On Error"
  N17:150/8  TIC401_DBA  "TIC-40-1 Tempered Oil No-2 1 = PV Within Deadband"
  N17:150/9  TIC401_UL  "TIC-40-1 Tempered Oil No-2 Output Greaater Than Upper CV"
  N17:150/10  TIC401_LL  "TIC-40-1 Tempered Oil No-2 Output Less Than Lower CV"
  N17:150/11  TIC401_SPA  "TIC-40-1 Tempered Oil No-2 Setpoint Out of Range"
  N17:150/12  TIC401_PVA  "TIC-40-1 Tempered Oil No-2 PV Out of Range"
  N17:150/13  TIC401_DN  "TIC-40-1 Tempered Oil No-2 PID Done"
  N17:150/15  TIC401_EN  "TIC-40-1 Tempered Oil No-2 PID Enabled"
  N17:151  TIC401_EC  "TIC-40-1 Tempered Oil No-2 PID Sub Error Code"
  N17:153  TIC401_G  "TIC-40-1 Tempered Oil No-2 Gain"
  N17:154  TIC401_TI  "TIC-40-1 Tempered Oil No-2 Reset"
  N17:155  TIC401_TD  "TIC-40-1 Tempered Oil No-2 Rate"
  N17:156  TIC401_FFD  "TIC-40-1 Tempered Oil No-2 Feed Forward Bias"
  N17:159  TIC401_DB  "TIC-40-1 Tempered Oil No-2 Deadband"
  N17:160  TIC401_C1  "TIC-40-1 Tempered Oil No-2 Used by PID Statement Do Not Alter"
  N17:161  TIC401_OMAX  "TIC-40-1 Tempered Oil No-2 Output Maximum"
  N17:162  TIC401_OMIN  "TIC-40-1 Tempered Oil No-2 Output Minimum"
  N17:163  TIC401_TIM  "TIC-40-1 Tempered Oil No-2 Last Loop Update Time"
  N17:165  TIC401_ERR  "TIC-40-1 Tempered Oil No-2 Scaled Error"
  N17:166  TIC401_OUT  "TIC-40-1 Tempered Oil No-2 Output 0/100%"
  N17:167  TIC401_C2  "TIC-40-1 Tempered Oil No-2 Used by PID Statement Do Not Alter"
  N17:168  TIC401_C3  "TIC-40-1 Tempered Oil No-2 Used by PID Statement Do Not Alter"
  N17:169  TIC401_C4  "TIC-40-1 Tempered Oil No-2 Used by PID Statement Do Not Alter"
  N17:170  TIC401_C5  "TIC-40-1 Tempered Oil No-2 Used by PID Statement Do Not Alter"
  N17:171  TIC401_C6  "TIC-40-1 Tempered Oil No-2 Used by PID Statement Do Not Alter"
  N17:172  TIC401_C7  "TIC-40-1 Tempered Oil No-2 Used by PID Statement Do Not Alter"
  N20:0  HMI_IFIX_JKT  "IFix and PanelView Jacket Fluids"
  N20:0/0  EV1_STM_OIL  "EV-1 Jacket Steam/Oil Select 0 = Oil 1 = Steam"
  N20:0/1  TK04_STM_TEMPWATER  "0 = Tempered Water 1 = Steam used on Feed Tank Graphic Jacket"
  N20:0/2  HE19_DISPLAY  "Ifix and PanelView HE-19 Display 0 = Off 1 = On"
  N20:0/3  EV2_STM_OIL  "EV-2 Jacket Steam/Oil Select 0 = Oil 1 = Steam"
  N20:0/4  EV20_STM_OIL  "EV-20 Jacket Steam/Oil Select 0 = Oil 1 = Steam"
  N20:0/5  EV42_STM_OIL  "EV-42 Jacket Steam/Oil Select 0 = Oil 1 = Steam"
  N20:1  HMI1_SCREEN  "HMI-1 PanelView in Process Area Actual Screen Currently Displayed"
  N20:2  HMI2_SCREEN  "HMI-2 PanelView in Conference Room Actual Screen Currently Displayed"
  N20:11  HMI1_SCREEN_TO_OPEN  "HMI-1 PanelView in Process Area Screen to be Displayed by PLC"
  N20:12  HMI2_SCREEN_TO_OPEN  "HMI-2 PanelView in Conference Room Screen to be Displayed by PLC"
  N20:21  HMI1_LOGIN_VALUE  "HMI-1 PanelView in Process Area Login 0 = Oper, 1 = Admin"
  N20:22  HMI2_LOGIN_VALUE  "HMI-2 PanelView in Conference Room Login 0 = Oper, 1 = Admin"
  N20:23  IFIX_LOGIN_VALUE  "iFIX System Login 0 = Oper, 1 = Admin"
  N20:30  FT_02_ALRM_SP
  N20:31  FT_05_ALRM_SP
  N20:32  FT_06_ALRM_SP
  N20:33  TE_02_ALRM_SP
  N20:34  TE_03_ALRM_SP
  N20:35  TE_30_ALRM_SP
  N20:36  TE_11_ALRM_SP
  N20:37  TE_24_ALRM_SP
  N23:4  TE_PTR_MAX  "Maximum Value for TE Pointer"
  N23:241  FIC211_LIT_PTR  "Level Transmitter Associated with FIC-21-1"
  N23:242  FIC212_LIT_PTR  "Level Transmitter Associated with FIC-21-2"
  N23:243  FIC213_LIT_PTR  "Level Transmitter Associated with FIC-21-3"
  N23:244  FIC214_LIT_PTR  "Level Transmitter Associated with FIC-21-4"
  N23:251  LIC221_FIT_PTR  "Flow Transmitter Associated with LIC-22-1"
  N23:252  LIC222_FIT_PTR  "Flow Transmitter Associated with LIC-22-2"
  N23:253  LIC223_FIT_PTR  "Flow Transmitter Associated with LIC-22-3"
  N24:41  AI_CURRENT_MAX_IE8  "Analog Input Maximum Value = 20 mA DC (From IE8 AI Module)"
  N25:1  TE29_36_BTW_WORD_1  "TE-29 thru TE-36 BTW Word 1"
  N25:2  TE29_36_BTW_WORD_2  "TE-29 thru TE-36 BTW Word 2"
  N25:3  TE29_36_BTW_WORD_3  "TE-29 thru TE-36 BTW Word 3"
  N25:6  TE29_36_BTR_WORD_1  "TE-29 thru TE-36 BTR Word 1"
  N25:7  TE29_36_BTR_WORD_2  "TE-29 thru TE-36 BTR Word 2"
  N25:8  TE29_36_BTR_WORD_3  "TE-29 thru TE-36 BTR Word 3"
  N25:10/15  MCC3_IE8_BTW_ENAB  "RIO Rack 2 Slot 3 Analog Input Module BTW Enable Bit"
  N25:11  MCC3_IE8_BTW_WORD_1  "RIO Rack 2 Slot 3 Analog Input Module BTW Word 1"
  N25:12  MCC3_IE8_BTW_WORD_2  "RIO Rack 2 Slot 3 Analog Input Module BTW Word 2"
  N25:16  MCC3_IE8_BTR_WORD_1  "RIO Rack 2 Slot 3 Analog Input Module BTR Word 1"
  N25:17  MCC3_IE8_BTR_WORD_2  "RIO Rack 2 Slot 3 Analog Input Module BTR Word 2"
  N25:21  MCC4_OE4_BTW_WORD_1  "RIO Rack 2 Slot 4 Analog Output Module BTW Word 1"
  N25:22  MCC4_OE4_BTW_WORD_2  "RIO Rack 2 Slot 4 Analog Output Module BTW Word 2"
  N25:25/15  MCC4_OE4_BTR_ENAB  "RIO Rack 2 Slot 4 Analog Output Module BTR Enable Bit"
  N25:26  MCC4_OE4_BTR_WORD_1  "RIO Rack 2 Slot 4 Analog Output Module BTR Word 1"
  N25:27  MCC4_OE4_BTR_WORD_2  "RIO Rack 2 Slot 4 Analog Output Module BTR Word 2"
  N25:31  MCC5_OE4_BTW_WORD_1  "RIO Rack 2 Slot 5 Analog Output Module BTW Word 1"
  N25:32  MCC5_OE4_BTW_WORD_2  "RIO Rack 2 Slot 5 Analog Output Module BTW Word 2"
  N25:35/15  MCC5_OE4_BTR_ENAB  "RIO Rack 2 Slot 5 Analog Output Module BTR Enable Bit"
  N25:36  MCC5_OE4_BTR_WORD_1  "RIO Rack 2 Slot 5 Analog Output Module BTR Word 1"
  N25:37  MCC5_OE4_BTR_WORD_2  "RIO Rack 2 Slot 5 Analog Output Module BTR Word 2"
  N25:100/12  PN5_IE81_BTW_ERROR
  N25:100/13  PN5_IE81_BTW_DONE
  N25:101  PN5_IE81_BTW_WORD_1  "RIO Rack 0 Slot 1 Analog Input Module BTW to Update Data to Outputs Word 1"
  N25:102  PN5_IE81_BTW_WORD_2  "RIO Rack 0 Slot 1 Analog Input Module BTW to Update Data to Outputs Word 2"
  N25:105/13  PN5_IE81_BTR_DONE
  N25:106  PN5_IE81_BTR_WORD_1  "RIO Rack 0 Slot 1 Analog Input Module BTR to Read Data Word 1"
  N25:107  PN5_IE81_BTR_WORD_2  "RIO Rack 0 Slot 1 Analog Input Module BTR to Read Data Word 2"
  N25:110/12  PN5_IE82_BTW_ERROR
  N25:110/13  PN5_IE82_BTW_DONE
  N25:111  PN5_IE82_BTW_WORD_1  "RIO Rack 0 Slot 2 Analog Input Module BTW to Update Data to Outputs Word 1"
  N25:112  PN5_IE82_BTW_WORD_2  "RIO Rack 0 Slot 2 Analog Input Module BTW to Update Data to Outputs Word 2"
  N25:115/13  PN5_IE82_BTR_DONE
  N25:116  PN5_IE82_BTR_WORD_1  "RIO Rack 0 Slot 2 Analog Input Module BTR to Read Data Word 1"
  N25:117  PN5_IE82_BTR_WORD_2  "RIO Rack 0 Slot 2 Analog Input Module BTR to Read Data Word 2"
  N25:121  PN5_OE41_BTW_WORD_1  "RIO Rack 0 Slot 3 Analog Output Module BTW to Update Data to Outputs Word 1"
  N25:122  PN5_OE41_BTW_WORD_2  "RIO Rack 0 Slot 3 Analog Output Module BTW to Update Data to Outputs Word 2"
  N25:125/15  PN5_OE41_BTR_ENAB
  N25:126  PN5_OE41_BTR_WORD_1  "RIO Rack 0 Slot 3 Analog Output Module BTR to Read Status of Outputs Word 1"
  N25:127  PN5_OE41_BTR_WORD_2  "RIO Rack 0 Slot 3 Analog Output Module BTR to Read Status of Outputs Word 2"
  N50:0  SS_01  "On/Off Selector Switch File 1 for all Devices"
  N50:1  SS_02  "On/Off Selector Switch File 2 for all Devices"
  N50:2  ILOCK_01  "Interlock File 1 for all Devices"
  N50:3  ILOCK_02  "Interlock File 2 for all Devices"
  N50:4  1SHOT_ON_O1  "1-Shot On File 1 For all Devices"
  N50:5  1SHOT_ON_02  "1-Shot On File 2 For all Devices"
  N50:6  1SHOT_OFF_01  "1-Shot Off File 1 For all Devices"
  N50:7  1SHOT_OFF_02  "1-Shot Off File 2 For all Devices"
  N50:8  OSR_ON_01  "OSR ON File 1 For all Devices"
  N50:9  OSR_ON_02  "OSR ON File 2 For all Devices"
  N50:10  OSR_OFF_01  "OSR OFF File 1 For all Devices"
  N50:11  OSR_OFF_02  "OSR OFF File 2 For all Devices"
  N50:13  VFD_MTR_RUN_BITS  "Run Bits as defined by selected VFD By Motor Tag"
  N50:14  VFD_MTR_ENABLE_BITS  "Enable CR Bits as defined by selected VFD By Motor Tag"
  N50:15  IFIX_PBS  "iFIX PB's"
  N50:16  IFIX_PB_1_SHOTS  "iFIX PB's 1-Shots"
  N50:17  IFIX_PB_OSRS  "iFIX PB's OSR's"
  N50:30/6  "Stop Auto IE8 Read"
  N50:30/7  "toggle IE8 Read"
  N61:2  VFD_RUN_BITS_2  "These Bits Initcate the UnderRange Status for the appropriate VFD"
  O:7.1  TE02_SET  "This File Determines Units (°C or °F) & Accuracy(0 or 0.0) for TE-2"
  O:7.2  TE03_SET  "This File Determines Units (°C or °F) & Accuracy(0 or 0.0) for TE-3"
  O:7.3  TE04_SET  "This File Determines Units (°C or °F) & Accuracy(0 or 0.0) for TE-4"
  O:8.0  TE05_SET  "This File Determines Units (°C or °F) & Accuracy(0 or 0.0) for TE-5"
  O:8.1  TE06_SET  "This File Determines Units (°C or °F) & Accuracy(0 or 0.0) for TE-6"
  O:8.2  TE07_SET  "This File Determines Units (°C or °F) & Accuracy(0 or 0.0) for TE-7"
  O:8.3  TE08_SET  "This File Determines Units (°C or °F) & Accuracy(0 or 0.0) for TE-8"
  O:9.1  TE10_SET  "This File Determines Units (°C or °F) & Accuracy(0 or 0.0) for TE-10"
  O:9.2  TE11_SET  "This File Determines Units (°C or °F) & Accuracy(0 or 0.0) for TE-11"
  O:9.3  TE12_SET  "This File Determines Units (°C or °F) & Accuracy(0 or 0.0) for TE-12"
  O:10.1  TE14_SET  "This File Determines Units (°C or °F) & Accuracy(0 or 0.0) for TE-14"
  O:10.2  TE15_SET  "This File Determines Units (°C or °F) & Accuracy(0 or 0.0) for TE-15"
  O:10.3  TE16_SET  "This File Determines Units (°C or °F) & Accuracy(0 or 0.0) for TE-16"
  O:11.1  TE18_SET  "This File Determines Units (°C or °F) & Accuracy(0 or 0.0) for TE-18"
  O:11.2  TE19_SET  "This File Determines Units (°C or °F) & Accuracy(0 or 0.0) for TE-19"
  O:11.3  TE20_SET  "This File Determines Units (°C or °F) & Accuracy(0 or 0.0) for TE-20"
  O:12.1  TE22_SET  "This File Determines Units (°C or °F) & Accuracy(0 or 0.0) for TE-22"
  O:12.2  TE23_SET  "This File Determines Units (°C or °F) & Accuracy(0 or 0.0) for TE-23"
  O:12.3  TE24_SET  "This File Determines Units (°C or °F) & Accuracy(0 or 0.0) for TE-24"
  O:18.1  TE26_SET  "This File Determines Units (°C or °F) & Accuracy(0 or 0.0) for TE-26"
  O:18.2  TE27_SET  "This File Determines Units (°C or °F) & Accuracy(0 or 0.0) for TE-27"
  O:18.3  TE28_SET  "This File Determines Units (°C or °F) & Accuracy(0 or 0.0) for TE-28"
  Q62:1  BYPASS_EH24_STOP  "Bypass EH-24 Stop Logic required to allow system to start EH-24 since no Run from External"
  Q64:1  BYPASS_EH27_STOP  "Bypass EH-27 Stop Logic required to allow system to start EH-27 since no Run from External"
  S:1/0  PLC_MODE  "Processor Mode Bit 0 0 = Run Mode 1 = Program Mode"
  T4:21.PRE  FT01_AVG_TIMER_SP  "FT-1 Average Timer Time Setpoint (Sec's)"
  T4:22.PRE  FT02_AVG_TIMER_SP  "FT-2 Average Timer Time Setpoint (Sec's)"
  T4:23.PRE  FT03_AVG_TIMER_SP  "FT-3 Average Timer Time Setpoint (Sec's)"
  T4:24.PRE  FT04_AVG_TIMER_SP  "FT-4 Average Timer Time Setpoint (Sec's)"
  T4:25.PRE  FT05_AVG_TIMER_SP  "FT-5 Average Timer Time Setpoint (Sec's)"
  T4:26.PRE  FT06_AVG_TIMER_SP  "FT-6 Average Timer Time Setpoint (Sec's)"
  T51:12  EH24_TIMER  "EH-24 Hot Oil Heater O.L. Timer"
  T51:51  ALARM_RK0_SL1_TMR  "Alarm Read or Write Fault RIO Rack 0 Slot 1 TImer"
  T51:52  ALARM_RK0_SL2_TMR  "Alarm Read or Write Fault RIO Rack 0 Slot 2 TImer"
  T51:53  ALARM_RK0_SL3_TMR  "Alarm Read or Write Fault RIO Rack 0 Slot 3 TImer"
  T51:54  ALARM_RK0_SL4_TMR  "Alarm Read or Write Fault RIO Rack 0 Slot 4 TImer"
  T51:55  ALARM_RK0_SL5_TMR  "Alarm Read or Write Fault RIO Rack 0 Slot 5 TImer"
  T51:56  ALARM_RK0_SL6_TMR  "Alarm Read or Write Fault RIO Rack 0 Slot 6 TImer"
  T51:57  ALARM_RK0_SL7_TMR  "Alarm Read or Write Fault RIO Rack 0 Slot 7 TImer"
  U:105  "FIC-46-1"
  U:106  "LIC-22-1-1"

COMMENTS NOT ATTACHED TO A CURRENT RUNG
  B3:0/0: This Rung Ensures that the Bit B3/0
    is always Off.
    It is used in the HMI displays as needed
  B3:5/1: This Rung Determines the Status of
    TAH-29-2
    Water To Sewer
    High Temp Alarm
    The Alarm is Set when the Temp Reaches the SP
    and will not be able to be reset until
    the Temp drops below the Reset SP
  B3:12/4: This Rung Determines the Status of
    FAL-24-1 Hot Oil Low Flow
    PAL-24-1 Hot Oil Low Pressure
    and
    PAH-24-1 Hot Oil High Pressure
    Alarms
  B3:15: This Rung Resets all Alarms
    when the operator presses the
    Alarm Reset PB on any HMI Terminal
  B223:0/1: This Rung Starts EV-2 Rotor Drive
    when the operator presses the EV-2 PB
    AND
    the Interlocks are satisfied and the motor is Off
  B223:0/2: This Rung Starts EV-3 Rotor Drive
    when the operator presses the EV-3 PB
    AND
    the Interlocks are satisfied and the motor is Off
  B223:0/3: This Rung Starts AG-4 Feed Tank Agitator
    when the operator presses the AG-4 PB
    AND
    the Interlocks are satisfied and the motor is Off
  B223:0/4: This Rung Starts VP-9 Beach-Ross Vacuum Pump
    when the operator presses the VP-9 PB
    AND
    the Interlocks are satisfied and the motor is Off
  B223:0/5: This Rung Starts VP-10 Kinney Vacuum Pump
    when the operator presses the VP-10 PB
    AND
    the Interlocks are satisfied and the motor is Off
  B223:0/6: This Rung Starts PU-11, Tempered Water Loop No-1 Pump
    when the operator presses the PU-11 PB
    AND
    the Interlocks are satisfied and the motor is Off
  B223:0/7: This Rung Starts PU-12, Tempered Water Loop No-2 Pump
    when the operator presses the PU-12 PB
    AND
    the Interlocks are satisfied and the motor is Off
  B223:0/8: This Rung Starts PU-15, Tempered Oil Loop No-1 Pump
    when the operator presses the PU-15 PB
    AND
    the Interlocks are satisfied and the motor is Off
  B223:0/9: This Rung Starts VB-35, TutHill Vacuum Blower
    when the operator presses the VB-35 PB
    AND
    the Interlocks are satisfied and the motor is Off
  B223:0/10: This Rung Starts PU-21, Feed Pump No-1
    when the operator presses the PU-21 PB
    AND
    the Interlocks are satisfied and the motor is Off
  B223:0/11: This Rung Starts PU-23 Hot Oil Pump
    when the operator presses the PU-23 PB (Local or HMI)
    AND the motor is Off
    OR
    The Interlocks are satisfied
  B223:0/12: This Rung Starts EH-24 Hot Oil Heater
    when the operator presses the EH-24 PB (Local or HMI)
    AND the Heater is Off
    OR
    The Interlocks are satisfied
  B223:0/13: This Rung Starts VB-26, Roots Vacuum Blower
    when the operator presses the VB-26 PB
    AND
    the Interlocks are satisfied and the motor is Off
  B223:0/15: This Rung Starts PU-30, Water Header Booster Pump
    when the operator presses the PU-30 PB
    AND
    the Interlocks are satisfied and the motor is Off
  B225:0/0: This Rung Starts PU-22, Feed Pump No-2
    when the operator presses the PU-22 PB
    AND
    the Interlocks are satisfied and the motor is Off
  B225:0/1: This Rung controls the status of
    EH-27 Contactor based on
    the whether EH-27 is enabled, and what the current
    TIC-24-1 PV & SPs are
  F21:[N110:0]: This Rung Converts the TE Integer Data to
    Floating Point (Real) by dividing the Integer value by 10.0
  F22:1: This Rung Moves the
    Selected Flow transmitter's
    Data to that for
    FT-1-1
  F22:2: This Rung Moves the
    Selected Flow transmitter's
    Data to that for
    FT-2-1
  F22:3: This Rung Moves the
    Selected Flow transmitter's
    Data to that for
    FT-3-1
  F22:14: This Rung Moves the
    Selected Flow transmitter's
    Data to that for
    PT-4-1
  F22:15: This Rung Moves the
    Selected Flow transmitter's
    Data to that for
    PT-5-1
  F22:16: This Rung Moves the
    Selected Flow transmitter's
    Data to that for
    PT-6-1
  F22:94: This Rung Moves the Selected TE's
    into the TE locations
    as shown below
  F22:143: This Rung Moves the Selected TE's
    into the TE locations
    as shown below
  F22:192: This Rung Moves the Selected TE's
    into the TE locations
    as shown below
  F22:211: This Rung moves the
    Selected FT values
    to FT-1-1 Value
  F22:217: This Rung Moves the Value of the Selected Flow Transmitter
    to FT-20-1, FT-20-2 and FT-20-3 Values
    Based on the Value of each's Pointer
  F28:0: This Rung Calculates the
    WY-1-1 Platform Scale No-1 Flow Rate in LBs/Hr
    Based on the change in weight over the last 30 Seconds
    Then Saves the current Value to be used in the next calculation
    Flow Rate is Based on Following Calc:
    
    Flow Rate = [(Last Weight) - (Current Weight)] * 120
    
    Absolute Value is used to Ignore Whether Weight is being Added or Removed from Scale
    (120 is number of 30 Second Intervals in 1 Hour)
  F29:8: This rung places
    FIC-21-1
    into Manual mode whenever PU-21
    is started or stopped.
    When Started, an initial SP is entered to start the Pump
    When Stopped, a value of 0 is entered to ensure the Pump does not run
    Auto Mode must be selected by the Operator
  F29:18: This rung places
    FIC-21-2
    into Manual mode whenever PU-21-2
    is started or stopped.
    When Started, an initial SP is entered to start the Pump
    When Stopped, a value of 0 is entered to ensure the Pump does not run
    Auto Mode must be selected by the Operator
  F29:44: This rung copies the
    PT-46-1 Data to
    PIC-46-1 Data (For use by iFIX)
  F29:188: This Rung Places
    TIC-24-1
    Hot Oil System
    Into Manual Mode with an output of 0% whenever EH-24 is stopped
    OR
    Into Auto Mode with an Initial Setpoint whenever EH-24 is started
  F30:5: This Rung Calculates the 25%, 50% & 75%
    Values for
    IT-2-1
    EV-2 Rotor Current
    Based on Minimum and Maximum Values
    Entered by Operator
    (For use on HMI Displays, etc)
  F30:45: This Rung Calculates the 25%, 50% & 75%
    Values for
    SY-3-1 Hp
    EV-3 Hp
    Based on Minimum and Maximum Values
    Entered by Operator
    (For use on HMI Displays, etc)
  F30:223: This Rung Calculates the 25%, 50% & 75%
    Values for
    LIT-1
    Based on Minimum and Maximum Values
    Entered by Operator
    (For use on HMI Displays, etc)
  F30:225: This Rung Converts the PID Integer value of
    LIC-1 PV
    to a Floating point Value used by the HMI's
  F30:229: This Rung Sets the Setpoint and Output for
    LIC-1
    Based on the Auto/Manual Mode of the Controller
    In Manual Mode, The Setpoint is set equal to the Process Variable - Both the Floating Point Value, and the PID Statement Value -
    (To allow bumpless transfer when Auto Mode is Selected)
    Also In Manual Mode The Output entered by the Operator is scaled to a value required by the PID Statement then Sent to the PID Output Value
    
    In Auto Mode, The Setpoint is Entered by the Operator from Any HMI terminal, Multiplied by 10, and placed in the PID Statement's Setpoint Location
    Also In Auto Mode, the Output (used by the Operator) is set equal to the actual value of the pID statement
    (To allow bumpless transfer when Manual Mode is Selected)
  F60:[N23:73]: For PU-21-3
    This Rung loads the OFF speed when stopped
    or
    The Initial Starting Speed when started
    If Running, the operator can adjust the running speed via the HMI's
    The speed is then moved to
    the sellected VFD's Speed Control register
    via the Scale Function
    to actually adjust the VFD's Speed
  I:6.19/4: This Rung Starts PU-13 Tempered Oil Pump No-2
    when the operator presses the PU-13 PB
    AND
    the Interlocks are satisfied and the motor is Off
  N13:40: This Rung Controls the Status and Speed of
    VFD05
    if it's controls are enabled
  N13:41: This Rung Controls the Status and Speed of
    VFD06
    if it's controls are enabled
  N13:42: This Rung Controls the Status and Speed of
    VFD07
    if it's controls are enabled
  N13:43: This Rung Controls the Status and Speed of
    VFD08
    if it's controls are enabled
  N15:2: This Rung Sets the Setpoint for
    FIC-21-1
    to the Minimum Setpoint Entered in the PID Statement
    if it is not within the acceptable range for the PID Statement.
    This is done to prevent the PLC from faulting
     should an invalid number result from either Operator Entry or when the FT used for FIC-21-1 Is changed
  N15:25: This Rung Reads the Status of the 1794-IE8 madc Output Module
    Located in Slot 4 of the Remote I/O Rack Data
    Located in the MCC area
  N15:32: This Rung Sets the Setpoint for
    FIC-22-1
    to the Minimum Setpoint Entered in the PID Statement
    if it is not within the acceptable range for the PID Statement.
    This is done to prevent the PLC from faulting
     should an invalid number result from either Operator Entry or when the FT used for FIC-22-1 Is changed
  N15:68: This Rung Moves the
    PT-5 Data to the
    PIC-9-1 PID Statement if the PIC-9-1 Pointer is1.
  N18:1: This Rung Places
    FIC-21-1
    into manual Mode, with an Output of 0
    When PU-21 is stopped
  N18:2: This Rung Places
    FIC-22-1
    into manual Mode, with an Output of 0
    When PU-22 is stopped
  N23:75: This rung checks the value of all
    FIC, EV amd AG Output Pointers which determine which VFD is used.
    If any are greater than the max value shown,
    OR
    The Hp of the motor is greater than that of the selected VFD
    it will be reset to 0
    to prevent PLC or VFD faults
  N23:80: This rung adds 1 to the value
    of the Max Number of VFDs Used.
    This Value is then used elsewhere in logic to determine if an illegal value has been assigned to to
    any motor that uses a VFD
  N23:91: This Rung Sets the
    VFD01 User Value
    to 0
    If none of the User Pointers are equal to 1
  N23:92: This Rung Sets the
    VFD02 User Value
    to 0
    If none of the User Pointers are equal to 2
  N23:93: This Rung Sets the
    VFD03 User Value
    to 0
    If none of the User Pointers are equal to 3
  N23:94: This Rung Sets the
    VFD04 User Value
    to 0
    If none of the User Pointers are equal to 4
  N23:95: This Rung Sets the
    VFD05 User Value
    to 0
    If none of the User Pointers are equal to 5
  N23:96: This Rung Sets the
    VFD06 User Value
    to 0
    If none of the User Pointers are equal to 6
  N23:97: This Rung Sets the
    VFD07 User Value
    to 0
    If none of the User Pointers are equal to 7
  N23:98: This Rung Sets the
    VFD01 thru VFD08
    User Value to 10 if any are assigned to FIC-21-1
    
